LIN {X 0,Y 162.207,Z 623.007,A -85,B 0,C 180,E1 -23497.47,E2 -23497.47} C_VEL
LIN {X 0,Y 162.719,Z 622.375,A -85,B 0,C 180,E1 -23499.95,E2 -23499.95} C_VEL
LIN {X 0,Y 163.523,Z 621.28,A -85,B 0,C 180,E1 -23502.411,E2 -23502.411} C_VEL
LIN {X 0,Y 165.346,Z 618.557,A -85,B 0,C 180,E1 -23506.04,E2 -23506.04} C_VEL
LIN {X 0,Y 167.897,Z 614.612,A -85,B 0,C 180,E1 -23509.566,E2 -23509.566} C_VEL
LIN {X 0,Y 168.435,Z 613.877,A -85,B 0,C 180,E1 -23510.136,E2 -23510.136} C_VEL
LIN {X 0,Y 170.028,Z 614.229,A -85,B 0,C 180,E1 -23511.925,E2 -23511.925} C_VEL
LIN {X 0,Y 175.274,Z 613.945,A -85,B 0,C 180,E1 -23516.173,E2 -23516.173} C_VEL
LIN {X 0,Y 178.341,Z 613.349,A -85,B 0,C 180,E1 -23518.223,E2 -23518.223} C_VEL
LIN {X 0,Y 183.249,Z 611.746,A -85,B 0,C 180,E1 -23520.885,E2 -23520.885} C_VEL
LIN {X 0,Y 185.044,Z 611.049,A -85,B 0,C 180,E1 -23521.95,E2 -23521.95} C_VEL
LIN {X 0,Y 186.792,Z 609.893,A -85,B 0,C 180,E1 -23523.665,E2 -23523.665} C_VEL
LIN {X 0,Y 188.276,Z 608.112,A -85,B 0,C 180,E1 -23526.659,E2 -23526.659} C_VEL
LIN {X 0,Y 190.28,Z 605.857,A -85,B 0,C 180,E1 -23530.266,E2 -23530.266} C_VEL
LIN {X 0,Y 191.354,Z 605.077,A -85,B 0,C 180,E1 -23531.385,E2 -23531.385} C_VEL
LIN {X 0,Y 192.086,Z 604.286,A -85,B 0,C 180,E1 -23532.966,E2 -23532.966} C_VEL
LIN {X 0,Y 192.613,Z 603.111,A -85,B 0,C 180,E1 -23536.867,E2 -23536.867} C_VEL
LIN {X 0,Y 192.568,Z 602.746,A -85,B 0,C 180,E1 -23540.035,E2 -23540.035} C_VEL
LIN {X 0,Y 192.239,Z 602.8,A -85,B 0,C 180,E1 -23541.575,E2 -23541.575} C_VEL
LIN {X 0,Y 191.24,Z 603.167,A -85,B 0,C 180,E1 -23543.985,E2 -23543.985} C_VEL
LIN {X 0,Y 188.877,Z 604.094,A -85,B 0,C 180,E1 -23546.073,E2 -23546.073} C_VEL
LIN {X 0,Y 184.48,Z 605.231,A -85,B 0,C 180,E1 -23547.768,E2 -23547.768} C_VEL
LIN {X 0,Y 176.516,Z 606.429,A -85,B 0,C 180,E1 -23551.46,E2 -23551.46} C_VEL
LIN {X 0,Y 171.67,Z 606.356,A -85,B 0,C 180,E1 -23554.248,E2 -23554.248} C_VEL
LIN {X 0,Y 166.772,Z 605.292,A -85,B 0,C 180,E1 -23557.712,E2 -23557.712} C_VEL
LIN {X 0,Y 164.167,Z 604.166,A -85,B 0,C 180,E1 -23559.972,E2 -23559.972} C_VEL
LIN {X 0,Y 159.875,Z 600.675,A -85,B 0,C 180,E1 -23564.707,E2 -23564.707} C_VEL
LIN {X 0,Y 157.891,Z 597.165,A -85,B 0,C 180,E1 -23568.315,E2 -23568.315} C_VEL
LIN {X 0,Y 156.697,Z 592.416,A -85,B 0,C 180,E1 -23572.267,E2 -23572.267} C_VEL
LIN {X 0,Y 156.112,Z 586.613,A -85,B 0,C 180,E1 -23576.128,E2 -23576.128} C_VEL
LIN {X 0,Y 156.043,Z 579.511,A -85,B 0,C 180,E1 -23580,E2 -23580} C_VEL
LIN {X 0,Y 156.277,Z 572.106,A -85,B 0,C 180,E1 -23583.223,E2 -23583.223} C_VEL
LIN {X 0,Y 156.781,Z 562.966,A -85,B 0,C 180,E1 -23586.435,E2 -23586.435} C_VEL
LIN {X 0,Y 156.964,Z 559.635,A -85,B 0,C 180,E1 -23587.477,E2 -23587.477} C_VEL
LIN {X 0,Y 156.789,Z 560.465,A -85,B 0,C 180,E1 -23587.728,E2 -23587.728} C_VEL
LIN {X 0,Y 158.13,Z 562.339,A -85,B 0,C 180,E1 -23589.28,E2 -23589.28} C_VEL
LIN {X 0,Y 160.819,Z 561.897,A -85,B 0,C 180,E1 -23590.717,E2 -23590.717} C_VEL
LIN {X 0,Y 163.892,Z 561.849,A -85,B 0,C 180,E1 -23592.381,E2 -23592.381} C_VEL
LIN {X 0,Y 168.567,Z 561.369,A -85,B 0,C 180,E1 -23594.487,E2 -23594.487} C_VEL
LIN {X 0,Y 172.959,Z 561.867,A -85,B 0,C 180,E1 -23596.525,E2 -23596.525} C_VEL
LIN {X 0,Y 175.402,Z 568.322,A -85,B 0,C 180,E1 -23599.303,E2 -23599.303} C_VEL
LIN {X 0,Y 175.617,Z 573.789,A -85,B 0,C 180,E1 -23601.111,E2 -23601.111} C_VEL
LIN {X 0,Y 175.037,Z 581.344,A -85,B 0,C 180,E1 -23603.673,E2 -23603.673} C_VEL
LIN {X 0,Y 174.064,Z 586.458,A -85,B 0,C 180,E1 -23605.485,E2 -23605.485} C_VEL
LIN {X 0,Y 170.852,Z 593.117,A -85,B 0,C 180,E1 -23607.82,E2 -23607.82} C_VEL
LIN {X 0,Y 167.861,Z 598.504,A -85,B 0,C 180,E1 -23610.16,E2 -23610.16} C_VEL
LIN {X 0,Y 164.679,Z 603.67,A -85,B 0,C 180,E1 -23613.039,E2 -23613.039} C_VEL
LIN {X 0,Y 161.608,Z 608.225,A -85,B 0,C 180,E1 -23616.436,E2 -23616.436} C_VEL
LIN {X 0,Y 159.378,Z 611.17,A -85,B 0,C 180,E1 -23619.492,E2 -23619.492} C_VEL
LIN {X 0,Y 157.997,Z 612.779,A -85,B 0,C 180,E1 -23621.854,E2 -23621.854} C_VEL
LIN {X 0,Y 156.118,Z 614.605,A -85,B 0,C 180,E1 -23626.077,E2 -23626.077} C_VEL
LIN {X 0,Y 154.878,Z 614.948,A -85,B 0,C 180,E1 -23630.557,E2 -23630.557} C_VEL
LIN {X 0,Y 154.344,Z 613.836,A -85,B 0,C 180,E1 -23635.047,E2 -23635.047} C_VEL
LIN {X 0,Y 154.333,Z 612.995,A -85,B 0,C 180,E1 -23636.874,E2 -23636.874} C_VEL
LIN {X 0,Y 154.603,Z 610.912,A -85,B 0,C 180,E1 -23639.996,E2 -23639.996} C_VEL
LIN {X 0,Y 155.155,Z 608.065,A -85,B 0,C 180,E1 -23643.064,E2 -23643.064} C_VEL
LIN {X 0,Y 156.072,Z 603.34,A -85,B 0,C 180,E1 -23646.794,E2 -23646.794} C_VEL
LIN {X 0,Y 157.166,Z 598.254,A -85,B 0,C 180,E1 -23649.894,E2 -23649.894} C_VEL
LIN {X 0,Y 158.396,Z 592.777,A -85,B 0,C 180,E1 -23652.571,E2 -23652.571} C_VEL
LIN {X 0,Y 160.251,Z 585.018,A -85,B 0,C 180,E1 -23655.611,E2 -23655.611} C_VEL
LIN {X 0,Y 162.014,Z 576.781,A -85,B 0,C 180,E1 -23658.108,E2 -23658.108} C_VEL
LIN {X 0,Y 162.751,Z 572.847,A -85,B 0,C 180,E1 -23659.109,E2 -23659.109} C_VEL
LIN {X 0,Y 162.183,Z 562.521,A -85,B 0,C 180,E1 -23661.589,E2 -23661.589} C_VEL
LIN {X 0,Y 161.198,Z 552.872,A -85,B 0,C 180,E1 -23663.427,E2 -23663.427} C_VEL
LIN {X 0,Y 159.728,Z 543.138,A -85,B 0,C 180,E1 -23664.95,E2 -23664.95} C_VEL
LIN {X 0,Y 157.671,Z 532.624,A -85,B 0,C 180,E1 -23666.325,E2 -23666.325} C_VEL
LIN {X 0,Y 158.334,Z 527.356,A -85,B 0,C 180,E1 -23671.27,E2 -23671.27} C_VEL
LIN {X 0,Y 157.895,Z 525.63,A -85,B 0,C 180,E1 -23673.188,E2 -23673.188} C_VEL
LIN {X 0,Y 157.826,Z 525.639,A -85,B 0,C 180,E1 -23677.676,E2 -23677.676} C_VEL
LIN {X 0,Y 157.707,Z 525.652,A -85,B 0,C 180,E1 -23681.361,E2 -23681.361} C_VEL
LIN {X 0,Y 157.479,Z 525.68,A -85,B 0,C 180,E1 -23685.53,E2 -23685.53} C_VEL
LIN {X 0,Y 157.37,Z 525.693,A -85,B 0,C 180,E1 -23690.931,E2 -23690.931} C_VEL
LIN {X 0,Y 157.315,Z 525.701,A -85,B 0,C 180,E1 -23696.684,E2 -23696.684} C_VEL
LIN {X 0,Y 157.278,Z 525.705,A -85,B 0,C 180,E1 -23702.425,E2 -23702.425} C_VEL
LIN {X 0,Y 157.317,Z 525.701,A -85,B 0,C 180,E1 -23706.473,E2 -23706.473} C_VEL
LIN {X 0,Y 157.274,Z 525.7,A -85,B 0,C 180,E1 -23712.088,E2 -23712.088} C_VEL
LIN {X 0,Y 157.3,Z 525.701,A -85,B 0,C 180,E1 -23715.63,E2 -23715.63} C_VEL
LIN {X 0,Y 157.285,Z 525.7,A -85,B 0,C 180,E1 -23721.276,E2 -23721.276} C_VEL
LIN {X 0,Y 157.29,Z 525.698,A -85,B 0,C 180,E1 -23724.488,E2 -23724.488} C_VEL
LIN {X 0,Y 157.291,Z 525.706,A -85,B 0,C 180,E1 -23728.095,E2 -23728.095} C_VEL
LIN {X 0,Y 157.319,Z 525.696,A -85,B 0,C 180,E1 -23733.465,E2 -23733.465} C_VEL
LIN {X 0,Y 157.392,Z 525.69,A -85,B 0,C 180,E1 -23739.667,E2 -23739.667} C_VEL
LIN {X 0,Y 157.476,Z 525.681,A -85,B 0,C 180,E1 -23744.468,E2 -23744.468} C_VEL
LIN {X 0,Y 157.77,Z 525.641,A -85,B 0,C 180,E1 -23749.736,E2 -23749.736} C_VEL
LIN {X 0,Y 157.822,Z 525.638,A -85,B 0,C 180,E1 -23752.323,E2 -23752.323} C_VEL
LIN {X 0,Y 158.256,Z 525.576,A -85,B 0,C 180,E1 -23760,E2 -23760} C_VEL
LIN {X 0,Y 157.822,Z 525.637,A -85,B 0,C 180,E1 -23767.677,E2 -23767.677} C_VEL
LIN {X 0,Y 157.703,Z 525.654,A -85,B 0,C 180,E1 -23771.362,E2 -23771.362} C_VEL
LIN {X 0,Y 157.476,Z 525.684,A -85,B 0,C 180,E1 -23775.532,E2 -23775.532} C_VEL
LIN {X 0,Y 157.367,Z 525.695,A -85,B 0,C 180,E1 -23780.933,E2 -23780.933} C_VEL
LIN {X 0,Y 157.312,Z 525.704,A -85,B 0,C 180,E1 -23786.685,E2 -23786.685} C_VEL
LIN {X 0,Y 157.276,Z 525.707,A -85,B 0,C 180,E1 -23792.427,E2 -23792.427} C_VEL
LIN {X 0,Y 157.281,Z 525.704,A -85,B 0,C 180,E1 -23796.458,E2 -23796.458} C_VEL
LIN {X 0,Y 157.23,Z 525.714,A -85,B 0,C 180,E1 -23802.104,E2 -23802.104} C_VEL
LIN {X 0,Y 157.323,Z 525.701,A -85,B 0,C 180,E1 -23807.928,E2 -23807.928} C_VEL
LIN {X 0,Y 157.937,Z 525.823,A -85,B 0,C 180,E1 -23814.498,E2 -23814.498} C_VEL
LIN {X 0,Y 158.756,Z 528.891,A -85,B 0,C 180,E1 -23816.218,E2 -23816.218} C_VEL
LIN {X 0,Y 158.764,Z 532.311,A -85,B 0,C 180,E1 -23817.915,E2 -23817.915} C_VEL
LIN {X 0,Y 158.394,Z 536.375,A -85,B 0,C 180,E1 -23819.811,E2 -23819.811} C_VEL
LIN {X 0,Y 160.336,Z 549.59,A -85,B 0,C 180,E1 -23821.175,E2 -23821.175} C_VEL
LIN {X 0,Y 161.128,Z 558.733,A -85,B 0,C 180,E1 -23822.41,E2 -23822.41} C_VEL
LIN {X 0,Y 161.352,Z 567.841,A -85,B 0,C 180,E1 -23823.926,E2 -23823.926} C_VEL
LIN {X 0,Y 161.312,Z 576.509,A -85,B 0,C 180,E1 -23825.715,E2 -23825.715} C_VEL
LIN {X 0,Y 160.941,Z 586.296,A -85,B 0,C 180,E1 -23828.213,E2 -23828.213} C_VEL
LIN {X 0,Y 159.369,Z 594.146,A -85,B 0,C 180,E1 -23830.688,E2 -23830.688} C_VEL
LIN {X 0,Y 157.885,Z 600.548,A -85,B 0,C 180,E1 -23833.183,E2 -23833.183} C_VEL
LIN {X 0,Y 156.793,Z 605.878,A -85,B 0,C 180,E1 -23835.729,E2 -23835.729} C_VEL
LIN {X 0,Y 155.929,Z 610.305,A -85,B 0,C 180,E1 -23838.299,E2 -23838.299} C_VEL
LIN {X 0,Y 155.113,Z 615.472,A -85,B 0,C 180,E1 -23842.189,E2 -23842.189} C_VEL
LIN {X 0,Y 154.855,Z 618.102,A -85,B 0,C 180,E1 -23844.793,E2 -23844.793} C_VEL
LIN {X 0,Y 154.815,Z 620.154,A -85,B 0,C 180,E1 -23847.399,E2 -23847.399} C_VEL
LIN {X 0,Y 154.892,Z 621.665,A -85,B 0,C 180,E1 -23850.001,E2 -23850.001} C_VEL
LIN {X 0,Y 154.775,Z 622.571,A -85,B 0,C 180,E1 -23852.604,E2 -23852.604} C_VEL
LIN {X 0,Y 154.857,Z 622.945,A -85,B 0,C 180,E1 -23855.209,E2 -23855.209} C_VEL
LIN {X 0,Y 155.172,Z 622.861,A -85,B 0,C 180,E1 -23857.811,E2 -23857.811} C_VEL
LIN {X 0,Y 155.715,Z 622.321,A -85,B 0,C 180,E1 -23860.402,E2 -23860.402} C_VEL
LIN {X 0,Y 156.597,Z 621.297,A -85,B 0,C 180,E1 -23862.969,E2 -23862.969} C_VEL
LIN {X 0,Y 158.528,Z 618.696,A -85,B 0,C 180,E1 -23866.749,E2 -23866.749} C_VEL
LIN {X 0,Y 161.228,Z 614.868,A -85,B 0,C 180,E1 -23870.411,E2 -23870.411} C_VEL
LIN {X 0,Y 162.615,Z 613.157,A -85,B 0,C 180,E1 -23871.887,E2 -23871.887} C_VEL
LIN {X 0,Y 166.021,Z 613.673,A -85,B 0,C 180,E1 -23875.046,E2 -23875.046} C_VEL
LIN {X 0,Y 168.934,Z 613.649,A -85,B 0,C 180,E1 -23877.235,E2 -23877.235} C_VEL
LIN {X 0,Y 175.704,Z 612.497,A -85,B 0,C 180,E1 -23881.333,E2 -23881.333} C_VEL
LIN {X 0,Y 179.68,Z 611.368,A -85,B 0,C 180,E1 -23883.203,E2 -23883.203} C_VEL
LIN {X 0,Y 183.551,Z 609.907,A -85,B 0,C 180,E1 -23885.054,E2 -23885.054} C_VEL
LIN {X 0,Y 186.575,Z 608.394,A -85,B 0,C 180,E1 -23887.065,E2 -23887.065} C_VEL
LIN {X 0,Y 189.284,Z 606.633,A -85,B 0,C 180,E1 -23889.14,E2 -23889.14} C_VEL
LIN {X 0,Y 190.28,Z 605.857,A -85,B 0,C 180,E1 -23890.266,E2 -23890.266} C_VEL
LIN {X 0,Y 190.856,Z 605.242,A -85,B 0,C 180,E1 -23891.41,E2 -23891.41} C_VEL
LIN {X 0,Y 190.445,Z 604.805,A -85,B 0,C 180,E1 -23893.173,E2 -23893.173} C_VEL
LIN {X 0,Y 189.135,Z 604.766,A -85,B 0,C 180,E1 -23894.933,E2 -23894.933} C_VEL
LIN {X 0,Y 186.189,Z 605.068,A -85,B 0,C 180,E1 -23898.626,E2 -23898.626} C_VEL
LIN {X 0,Y 185.854,Z 605.035,A -85,B 0,C 180,E1 -23899.895,E2 -23899.895} C_VEL
LIN {X 0,Y 184.79,Z 605.138,A -85,B 0,C 180,E1 -23903.006,E2 -23903.006} C_VEL
LIN {X 0,Y 182.966,Z 605.531,A -85,B 0,C 180,E1 -23904.818,E2 -23904.818} C_VEL
LIN {X 0,Y 174.336,Z 606.945,A -85,B 0,C 180,E1 -23908.395,E2 -23908.395} C_VEL
LIN {X 0,Y 166.248,Z 606.681,A -85,B 0,C 180,E1 -23912.596,E2 -23912.596} C_VEL
LIN {X 0,Y 163.292,Z 606.167,A -85,B 0,C 180,E1 -23914.508,E2 -23914.508} C_VEL
LIN {X 0,Y 157.542,Z 603.712,A -85,B 0,C 180,E1 -23919.091,E2 -23919.091} C_VEL
LIN {X 0,Y 154.115,Z 600.908,A -85,B 0,C 180,E1 -23922.758,E2 -23922.758} C_VEL
LIN {X 0,Y 151.609,Z 597.215,A -85,B 0,C 180,E1 -23926.598,E2 -23926.598} C_VEL
LIN {X 0,Y 150.168,Z 592.578,A -85,B 0,C 180,E1 -23930.572,E2 -23930.572} C_VEL
LIN {X 0,Y 149.434,Z 586.884,A -85,B 0,C 180,E1 -23934.603,E2 -23934.603} C_VEL
LIN {X 0,Y 149.186,Z 579.766,A -85,B 0,C 180,E1 -23938.651,E2 -23938.651} C_VEL
LIN {X 0,Y 149.403,Z 572.526,A -85,B 0,C 180,E1 -23942.022,E2 -23942.022} C_VEL
LIN {X 0,Y 149.647,Z 565.842,A -85,B 0,C 180,E1 -23944.63,E2 -23944.63} C_VEL
LIN {X 0,Y 149.485,Z 567.428,A -85,B 0,C 180,E1 -23945.396,E2 -23945.396} C_VEL
LIN {X 0,Y 152.87,Z 567.395,A -85,B 0,C 180,E1 -23947.928,E2 -23947.928} C_VEL
LIN {X 0,Y 155.992,Z 568.381,A -85,B 0,C 180,E1 -23950.382,E2 -23950.382} C_VEL
LIN {X 0,Y 164.946,Z 567.632,A -85,B 0,C 180,E1 -23954.812,E2 -23954.812} C_VEL
LIN {X 0,Y 168.848,Z 568.796,A -85,B 0,C 180,E1 -23956.94,E2 -23956.94} C_VEL
LIN {X 0,Y 170.034,Z 572.646,A -85,B 0,C 180,E1 -23958.683,E2 -23958.683} C_VEL
LIN {X 0,Y 169.597,Z 579.862,A -85,B 0,C 180,E1 -23961.26,E2 -23961.26} C_VEL
LIN {X 0,Y 168.174,Z 587.363,A -85,B 0,C 180,E1 -23964.13,E2 -23964.13} C_VEL
LIN {X 0,Y 164.933,Z 593.81,A -85,B 0,C 180,E1 -23966.51,E2 -23966.51} C_VEL
LIN {X 0,Y 161.238,Z 599.946,A -85,B 0,C 180,E1 -23969.334,E2 -23969.334} C_VEL
LIN {X 0,Y 157.228,Z 605.949,A -85,B 0,C 180,E1 -23973.056,E2 -23973.056} C_VEL
LIN {X 0,Y 154.425,Z 609.605,A -85,B 0,C 180,E1 -23976.274,E2 -23976.274} C_VEL
LIN {X 0,Y 152.748,Z 611.555,A -85,B 0,C 180,E1 -23978.538,E2 -23978.538} C_VEL
LIN {X 0,Y 150.822,Z 613.566,A -85,B 0,C 180,E1 -23981.79,E2 -23981.79} C_VEL
LIN {X 0,Y 149.331,Z 614.771,A -85,B 0,C 180,E1 -23985.092,E2 -23985.092} C_VEL
LIN {X 0,Y 147.999,Z 615.206,A -85,B 0,C 180,E1 -23989.446,E2 -23989.446} C_VEL
LIN {X 0,Y 147.303,Z 614.173,A -85,B 0,C 180,E1 -23994.203,E2 -23994.203} C_VEL
LIN {X 0,Y 147.373,Z 611.609,A -85,B 0,C 180,E1 -23999.137,E2 -23999.137} C_VEL
LIN {X 0,Y 148.04,Z 608.225,A -85,B 0,C 180,E1 -24003.026,E2 -24003.026} C_VEL
LIN {X 0,Y 149.03,Z 603.251,A -85,B 0,C 180,E1 -24007.103,E2 -24007.103} C_VEL
LIN {X 0,Y 150.148,Z 598.211,A -85,B 0,C 180,E1 -24010.283,E2 -24010.283} C_VEL
LIN {X 0,Y 151.466,Z 592.563,A -85,B 0,C 180,E1 -24013.141,E2 -24013.141} C_VEL
LIN {X 0,Y 153.372,Z 584.895,A -85,B 0,C 180,E1 -24016.242,E2 -24016.242} C_VEL
LIN {X 0,Y 155.287,Z 576.297,A -85,B 0,C 180,E1 -24018.909,E2 -24018.909} C_VEL
LIN {X 0,Y 155.824,Z 572.513,A -85,B 0,C 180,E1 -24019.933,E2 -24019.933} C_VEL
LIN {X 0,Y 155.241,Z 561.98,A -85,B 0,C 180,E1 -24022.52,E2 -24022.52} C_VEL
LIN {X 0,Y 154.221,Z 552.27,A -85,B 0,C 180,E1 -24024.442,E2 -24024.442} C_VEL
LIN {X 0,Y 152.614,Z 541.928,A -85,B 0,C 180,E1 -24026.12,E2 -24026.12} C_VEL
LIN {X 0,Y 150.798,Z 532.806,A -85,B 0,C 180,E1 -24027.327,E2 -24027.327} C_VEL
LIN {X 0,Y 151.343,Z 528.659,A -85,B 0,C 180,E1 -24031.329,E2 -24031.329} C_VEL
LIN {X 0,Y 150.826,Z 526.51,A -85,B 0,C 180,E1 -24033.672,E2 -24033.672} C_VEL
LIN {X 0,Y 150.765,Z 526.519,A -85,B 0,C 180,E1 -24038.038,E2 -24038.038} C_VEL
LIN {X 0,Y 150.636,Z 526.533,A -85,B 0,C 180,E1 -24041.545,E2 -24041.545} C_VEL
LIN {X 0,Y 150.384,Z 526.564,A -85,B 0,C 180,E1 -24046.283,E2 -24046.283} C_VEL
LIN {X 0,Y 150.351,Z 526.567,A -85,B 0,C 180,E1 -24050.791,E2 -24050.791} C_VEL
LIN {X 0,Y 150.244,Z 526.581,A -85,B 0,C 180,E1 -24057.281,E2 -24057.281} C_VEL
LIN {X 0,Y 150.218,Z 526.584,A -85,B 0,C 180,E1 -24062.633,E2 -24062.633} C_VEL
LIN {X 0,Y 150.223,Z 526.584,A -85,B 0,C 180,E1 -24067.457,E2 -24067.457} C_VEL
LIN {X 0,Y 150.21,Z 526.582,A -85,B 0,C 180,E1 -24071.53,E2 -24071.53} C_VEL
LIN {X 0,Y 150.249,Z 526.578,A -85,B 0,C 180,E1 -24075.441,E2 -24075.441} C_VEL
LIN {X 0,Y 150.228,Z 526.582,A -85,B 0,C 180,E1 -24079.084,E2 -24079.084} C_VEL
LIN {X 0,Y 150.234,Z 526.572,A -85,B 0,C 180,E1 -24082.678,E2 -24082.678} C_VEL
LIN {X 0,Y 150.215,Z 526.584,A -85,B 0,C 180,E1 -24087.365,E2 -24087.365} C_VEL
LIN {X 0,Y 150.242,Z 526.576,A -85,B 0,C 180,E1 -24092.717,E2 -24092.717} C_VEL
LIN {X 0,Y 150.349,Z 526.567,A -85,B 0,C 180,E1 -24099.207,E2 -24099.207} C_VEL
LIN {X 0,Y 150.381,Z 526.565,A -85,B 0,C 180,E1 -24103.715,E2 -24103.715} C_VEL
LIN {X 0,Y 150.687,Z 526.521,A -85,B 0,C 180,E1 -24109.248,E2 -24109.248} C_VEL
LIN {X 0,Y 150.761,Z 526.519,A -85,B 0,C 180,E1 -24111.961,E2 -24111.961} C_VEL
LIN {X 0,Y 151.216,Z 526.452,A -85,B 0,C 180,E1 -24120,E2 -24120} C_VEL
LIN {X 0,Y 150.761,Z 526.518,A -85,B 0,C 180,E1 -24128.039,E2 -24128.039} C_VEL
LIN {X 0,Y 150.632,Z 526.534,A -85,B 0,C 180,E1 -24131.546,E2 -24131.546} C_VEL
LIN {X 0,Y 150.38,Z 526.564,A -85,B 0,C 180,E1 -24136.284,E2 -24136.284} C_VEL
LIN {X 0,Y 150.348,Z 526.57,A -85,B 0,C 180,E1 -24140.793,E2 -24140.793} C_VEL
LIN {X 0,Y 150.242,Z 526.586,A -85,B 0,C 180,E1 -24147.283,E2 -24147.283} C_VEL
LIN {X 0,Y 150.216,Z 526.586,A -85,B 0,C 180,E1 -24152.635,E2 -24152.635} C_VEL
LIN {X 0,Y 150.209,Z 526.585,A -85,B 0,C 180,E1 -24157.462,E2 -24157.462} C_VEL
LIN {X 0,Y 150.168,Z 526.592,A -85,B 0,C 180,E1 -24161.514,E2 -24161.514} C_VEL
LIN {X 0,Y 150.189,Z 526.59,A -85,B 0,C 180,E1 -24165.421,E2 -24165.421} C_VEL
LIN {X 0,Y 150.332,Z 526.572,A -85,B 0,C 180,E1 -24169.12,E2 -24169.12} C_VEL
LIN {X 0,Y 150.773,Z 526.721,A -85,B 0,C 180,E1 -24173.538,E2 -24173.538} C_VEL
LIN {X 0,Y 151.819,Z 529.881,A -85,B 0,C 180,E1 -24175.455,E2 -24175.455} C_VEL
LIN {X 0,Y 151.937,Z 533.352,A -85,B 0,C 180,E1 -24177.307,E2 -24177.307} C_VEL
LIN {X 0,Y 151.634,Z 536.634,A -85,B 0,C 180,E1 -24178.833,E2 -24178.833} C_VEL
LIN {X 0,Y 153.5,Z 549.179,A -85,B 0,C 180,E1 -24180.19,E2 -24180.19} C_VEL
LIN {X 0,Y 154.308,Z 558.245,A -85,B 0,C 180,E1 -24181.477,E2 -24181.477} C_VEL
LIN {X 0,Y 154.489,Z 566.777,A -85,B 0,C 180,E1 -24182.942,E2 -24182.942} C_VEL
LIN {X 0,Y 154.475,Z 575.328,A -85,B 0,C 180,E1 -24184.756,E2 -24184.756} C_VEL
LIN {X 0,Y 154.186,Z 583.468,A -85,B 0,C 180,E1 -24186.852,E2 -24186.852} C_VEL
LIN {X 0,Y 153.763,Z 588.024,A -85,B 0,C 180,E1 -24188.202,E2 -24188.202} C_VEL
LIN {X 0,Y 152.226,Z 594.656,A -85,B 0,C 180,E1 -24190.446,E2 -24190.446} C_VEL
LIN {X 0,Y 150.759,Z 600.942,A -85,B 0,C 180,E1 -24193.062,E2 -24193.062} C_VEL
LIN {X 0,Y 149.64,Z 606.165,A -85,B 0,C 180,E1 -24195.727,E2 -24195.727} C_VEL
LIN {X 0,Y 148.601,Z 611.45,A -85,B 0,C 180,E1 -24199.097,E2 -24199.097} C_VEL
LIN {X 0,Y 148.06,Z 614.836,A -85,B 0,C 180,E1 -24201.815,E2 -24201.815} C_VEL
LIN {X 0,Y 147.79,Z 617.574,A -85,B 0,C 180,E1 -24204.544,E2 -24204.544} C_VEL
LIN {X 0,Y 147.719,Z 619.902,A -85,B 0,C 180,E1 -24207.581,E2 -24207.581} C_VEL
LIN {X 0,Y 147.796,Z 621.288,A -85,B 0,C 180,E1 -24210.001,E2 -24210.001} C_VEL
LIN {X 0,Y 147.695,Z 622.238,A -85,B 0,C 180,E1 -24212.729,E2 -24212.729} C_VEL
LIN {X 0,Y 147.792,Z 622.705,A -85,B 0,C 180,E1 -24215.459,E2 -24215.459} C_VEL
LIN {X 0,Y 148.119,Z 622.714,A -85,B 0,C 180,E1 -24218.185,E2 -24218.185} C_VEL
LIN {X 0,Y 148.734,Z 622.269,A -85,B 0,C 180,E1 -24220.896,E2 -24220.896} C_VEL
LIN {X 0,Y 149.694,Z 621.277,A -85,B 0,C 180,E1 -24223.578,E2 -24223.578} C_VEL
LIN {X 0,Y 151.743,Z 618.862,A -85,B 0,C 180,E1 -24227.522,E2 -24227.522} C_VEL
LIN {X 0,Y 154.597,Z 615.157,A -85,B 0,C 180,E1 -24231.328,E2 -24231.328} C_VEL
LIN {X 0,Y 156.803,Z 612.376,A -85,B 0,C 180,E1 -24233.616,E2 -24233.616} C_VEL
LIN {X 0,Y 162.686,Z 613.083,A -85,B 0,C 180,E1 -24238.374,E2 -24238.374} C_VEL
LIN {X 0,Y 165.992,Z 613.004,A -85,B 0,C 180,E1 -24240.537,E2 -24240.537} C_VEL
LIN {X 0,Y 173.805,Z 611.628,A -85,B 0,C 180,E1 -24244.481,E2 -24244.481} C_VEL
LIN {X 0,Y 177.724,Z 610.529,A -85,B 0,C 180,E1 -24246.383,E2 -24246.383} C_VEL
LIN {X 0,Y 182.416,Z 608.388,A -85,B 0,C 180,E1 -24249.597,E2 -24249.597} C_VEL
LIN {X 0,Y 183.587,Z 607.718,A -85,B 0,C 180,E1 -24250.786,E2 -24250.786} C_VEL
LIN {X 0,Y 185.295,Z 606.516,A -85,B 0,C 180,E1 -24253.058,E2 -24253.058} C_VEL
LIN {X 0,Y 185.911,Z 605.372,A -85,B 0,C 180,E1 -24257.121,E2 -24257.121} C_VEL
LIN {X 0,Y 185.854,Z 605.035,A -85,B 0,C 180,E1 -24259.895,E2 -24259.895} C_VEL
LIN {X 0,Y 185.169,Z 605.186,A -85,B 0,C 180,E1 -24260.858,E2 -24260.858} C_VEL
LIN {X 0,Y 182.748,Z 605.725,A -85,B 0,C 180,E1 -24262.057,E2 -24262.057} C_VEL
LIN {X 0,Y 176.733,Z 606.906,A -85,B 0,C 180,E1 -24263.881,E2 -24263.881} C_VEL
LIN {X 0,Y 172.841,Z 607.378,A -85,B 0,C 180,E1 -24265.235,E2 -24265.235} C_VEL
LIN {X 0,Y 164.22,Z 607.472,A -85,B 0,C 180,E1 -24269.099,E2 -24269.099} C_VEL
LIN {X 0,Y 160.388,Z 606.91,A -85,B 0,C 180,E1 -24271.184,E2 -24271.184} C_VEL
LIN {X 0,Y 153.763,Z 604.776,A -85,B 0,C 180,E1 -24275.71,E2 -24275.71} C_VEL
LIN {X 0,Y 148.558,Z 601.086,A -85,B 0,C 180,E1 -24280.661,E2 -24280.661} C_VEL
LIN {X 0,Y 145.567,Z 597.317,A -85,B 0,C 180,E1 -24284.601,E2 -24284.601} C_VEL
LIN {X 0,Y 143.733,Z 592.677,A -85,B 0,C 180,E1 -24288.721,E2 -24288.721} C_VEL
LIN {X 0,Y 142.701,Z 585.937,A -85,B 0,C 180,E1 -24293.638,E2 -24293.638} C_VEL
LIN {X 0,Y 142.399,Z 578.623,A -85,B 0,C 180,E1 -24297.879,E2 -24297.879} C_VEL
LIN {X 0,Y 142.586,Z 571.267,A -85,B 0,C 180,E1 -24301.412,E2 -24301.412} C_VEL
LIN {X 0,Y 142.309,Z 572.695,A -85,B 0,C 180,E1 -24302.123,E2 -24302.123} C_VEL
LIN {X 0,Y 142.597,Z 573.283,A -85,B 0,C 180,E1 -24302.825,E2 -24302.825} C_VEL
LIN {X 0,Y 149.166,Z 573.401,A -85,B 0,C 180,E1 -24308.332,E2 -24308.332} C_VEL
LIN {X 0,Y 152.028,Z 574.208,A -85,B 0,C 180,E1 -24310.656,E2 -24310.656} C_VEL
LIN {X 0,Y 160.894,Z 573.677,A -85,B 0,C 180,E1 -24315.194,E2 -24315.194} C_VEL
LIN {X 0,Y 164.234,Z 575.396,A -85,B 0,C 180,E1 -24317.431,E2 -24317.431} C_VEL
LIN {X 0,Y 164.21,Z 578.6,A -85,B 0,C 180,E1 -24318.724,E2 -24318.724} C_VEL
LIN {X 0,Y 163.125,Z 585.576,A -85,B 0,C 180,E1 -24321.482,E2 -24321.482} C_VEL
LIN {X 0,Y 161.692,Z 590.106,A -85,B 0,C 180,E1 -24323.358,E2 -24323.358} C_VEL
LIN {X 0,Y 157.075,Z 597.881,A -85,B 0,C 180,E1 -24326.579,E2 -24326.579} C_VEL
LIN {X 0,Y 153.408,Z 603.104,A -85,B 0,C 180,E1 -24329.488,E2 -24329.488} C_VEL
LIN {X 0,Y 150.18,Z 607.326,A -85,B 0,C 180,E1 -24332.609,E2 -24332.609} C_VEL
LIN {X 0,Y 147.386,Z 610.581,A -85,B 0,C 180,E1 -24335.84,E2 -24335.84} C_VEL
LIN {X 0,Y 145.051,Z 612.948,A -85,B 0,C 180,E1 -24339.172,E2 -24339.172} C_VEL
LIN {X 0,Y 142.77,Z 614.807,A -85,B 0,C 180,E1 -24343.564,E2 -24343.564} C_VEL
LIN {X 0,Y 141.147,Z 615.437,A -85,B 0,C 180,E1 -24348.321,E2 -24348.321} C_VEL
LIN {X 0,Y 140.263,Z 614.499,A -85,B 0,C 180,E1 -24353.292,E2 -24353.292} C_VEL
LIN {X 0,Y 140.216,Z 612.059,A -85,B 0,C 180,E1 -24358.44,E2 -24358.44} C_VEL
LIN {X 0,Y 140.995,Z 608.003,A -85,B 0,C 180,E1 -24363.344,E2 -24363.344} C_VEL
LIN {X 0,Y 141.967,Z 603.235,A -85,B 0,C 180,E1 -24367.387,E2 -24367.387} C_VEL
LIN {X 0,Y 143.433,Z 596.967,A -85,B 0,C 180,E1 -24371.427,E2 -24371.427} C_VEL
LIN {X 0,Y 145.371,Z 589.045,A -85,B 0,C 180,E1 -24375.219,E2 -24375.219} C_VEL
LIN {X 0,Y 146.893,Z 582.888,A -85,B 0,C 180,E1 -24377.566,E2 -24377.566} C_VEL
LIN {X 0,Y 148.575,Z 575.782,A -85,B 0,C 180,E1 -24379.781,E2 -24379.781} C_VEL
LIN {X 0,Y 148.877,Z 572.166,A -85,B 0,C 180,E1 -24380.831,E2 -24380.831} C_VEL
LIN {X 0,Y 148.337,Z 561.441,A -85,B 0,C 180,E1 -24383.538,E2 -24383.538} C_VEL
LIN {X 0,Y 147.291,Z 551.674,A -85,B 0,C 180,E1 -24385.552,E2 -24385.552} C_VEL
LIN {X 0,Y 145.834,Z 542.262,A -85,B 0,C 180,E1 -24387.15,E2 -24387.15} C_VEL
LIN {X 0,Y 143.943,Z 532.86,A -85,B 0,C 180,E1 -24388.512,E2 -24388.512} C_VEL
LIN {X 0,Y 144.349,Z 529.994,A -85,B 0,C 180,E1 -24391.394,E2 -24391.394} C_VEL
LIN {X 0,Y 143.709,Z 527.398,A -85,B 0,C 180,E1 -24394.381,E2 -24394.381} C_VEL
LIN {X 0,Y 143.686,Z 527.401,A -85,B 0,C 180,E1 -24398.436,E2 -24398.436} C_VEL
LIN {X 0,Y 143.572,Z 527.413,A -85,B 0,C 180,E1 -24401.756,E2 -24401.756} C_VEL
LIN {X 0,Y 143.317,Z 527.444,A -85,B 0,C 180,E1 -24407.11,E2 -24407.11} C_VEL
LIN {X 0,Y 143.277,Z 527.448,A -85,B 0,C 180,E1 -24411.253,E2 -24411.253} C_VEL
LIN {X 0,Y 143.19,Z 527.461,A -85,B 0,C 180,E1 -24417.936,E2 -24417.936} C_VEL
LIN {X 0,Y 143.169,Z 527.461,A -85,B 0,C 180,E1 -24423.435,E2 -24423.435} C_VEL
LIN {X 0,Y 143.107,Z 527.471,A -85,B 0,C 180,E1 -24429.673,E2 -24429.673} C_VEL
LIN {X 0,Y 143.154,Z 527.456,A -85,B 0,C 180,E1 -24433.416,E2 -24433.416} C_VEL
LIN {X 0,Y 143.155,Z 527.465,A -85,B 0,C 180,E1 -24437.424,E2 -24437.424} C_VEL
LIN {X 0,Y 143.137,Z 527.459,A -85,B 0,C 180,E1 -24441.773,E2 -24441.773} C_VEL
LIN {X 0,Y 143.183,Z 527.46,A -85,B 0,C 180,E1 -24447.321,E2 -24447.321} C_VEL
LIN {X 0,Y 143.188,Z 527.457,A -85,B 0,C 180,E1 -24452.062,E2 -24452.062} C_VEL
LIN {X 0,Y 143.275,Z 527.448,A -85,B 0,C 180,E1 -24458.745,E2 -24458.745} C_VEL
LIN {X 0,Y 143.314,Z 527.443,A -85,B 0,C 180,E1 -24462.888,E2 -24462.888} C_VEL
LIN {X 0,Y 143.6,Z 527.403,A -85,B 0,C 180,E1 -24468.71,E2 -24468.71} C_VEL
LIN {X 0,Y 143.682,Z 527.399,A -85,B 0,C 180,E1 -24471.562,E2 -24471.562} C_VEL
LIN {X 0,Y 144.175,Z 527.329,A -85,B 0,C 180,E1 -24480,E2 -24480} C_VEL
LIN {X 0,Y 143.682,Z 527.399,A -85,B 0,C 180,E1 -24488.438,E2 -24488.438} C_VEL
LIN {X 0,Y 143.569,Z 527.413,A -85,B 0,C 180,E1 -24491.758,E2 -24491.758} C_VEL
LIN {X 0,Y 143.314,Z 527.445,A -85,B 0,C 180,E1 -24497.111,E2 -24497.111} C_VEL
LIN {X 0,Y 143.274,Z 527.452,A -85,B 0,C 180,E1 -24501.255,E2 -24501.255} C_VEL
LIN {X 0,Y 143.188,Z 527.463,A -85,B 0,C 180,E1 -24507.938,E2 -24507.938} C_VEL
LIN {X 0,Y 143.166,Z 527.466,A -85,B 0,C 180,E1 -24513.436,E2 -24513.436} C_VEL
LIN {X 0,Y 143.08,Z 527.477,A -85,B 0,C 180,E1 -24519.684,E2 -24519.684} C_VEL
LIN {X 0,Y 143.104,Z 527.475,A -85,B 0,C 180,E1 -24523.437,E2 -24523.437} C_VEL
LIN {X 0,Y 143.176,Z 527.463,A -85,B 0,C 180,E1 -24527.416,E2 -24527.416} C_VEL
LIN {X 0,Y 143.519,Z 527.447,A -85,B 0,C 180,E1 -24532.39,E2 -24532.39} C_VEL
LIN {X 0,Y 145.063,Z 532.182,A -85,B 0,C 180,E1 -24535.448,E2 -24535.448} C_VEL
LIN {X 0,Y 144.951,Z 535.755,A -85,B 0,C 180,E1 -24537.419,E2 -24537.419} C_VEL
LIN {X 0,Y 144.856,Z 536.3,A -85,B 0,C 180,E1 -24537.703,E2 -24537.703} C_VEL
LIN {X 0,Y 146.704,Z 549.038,A -85,B 0,C 180,E1 -24539.154,E2 -24539.154} C_VEL
LIN {X 0,Y 147.569,Z 558.398,A -85,B 0,C 180,E1 -24540.567,E2 -24540.567} C_VEL
LIN {X 0,Y 147.691,Z 568.121,A -85,B 0,C 180,E1 -24542.359,E2 -24542.359} C_VEL
LIN {X 0,Y 147.572,Z 576.358,A -85,B 0,C 180,E1 -24544.244,E2 -24544.244} C_VEL
LIN {X 0,Y 147.128,Z 585.664,A -85,B 0,C 180,E1 -24546.839,E2 -24546.839} C_VEL
LIN {X 0,Y 145.987,Z 591.658,A -85,B 0,C 180,E1 -24548.836,E2 -24548.836} C_VEL
LIN {X 0,Y 143.937,Z 599.924,A -85,B 0,C 180,E1 -24552.233,E2 -24552.233} C_VEL
LIN {X 0,Y 142.767,Z 605.292,A -85,B 0,C 180,E1 -24555.024,E2 -24555.024} C_VEL
LIN {X 0,Y 141.624,Z 610.7,A -85,B 0,C 180,E1 -24558.552,E2 -24558.552} C_VEL
LIN {X 0,Y 141.029,Z 614.201,A -85,B 0,C 180,E1 -24561.403,E2 -24561.403} C_VEL
LIN {X 0,Y 140.642,Z 618.178,A -85,B 0,C 180,E1 -24565.703,E2 -24565.703} C_VEL
LIN {X 0,Y 140.652,Z 619.73,A -85,B 0,C 180,E1 -24567.925,E2 -24567.925} C_VEL
LIN {X 0,Y 140.717,Z 620.866,A -85,B 0,C 180,E1 -24570.001,E2 -24570.001} C_VEL
LIN {X 0,Y 140.618,Z 621.899,A -85,B 0,C 180,E1 -24572.866,E2 -24572.866} C_VEL
LIN {X 0,Y 140.721,Z 622.462,A -85,B 0,C 180,E1 -24575.734,E2 -24575.734} C_VEL
LIN {X 0,Y 141.082,Z 622.571,A -85,B 0,C 180,E1 -24578.596,E2 -24578.596} C_VEL
LIN {X 0,Y 141.753,Z 622.189,A -85,B 0,C 180,E1 -24581.44,E2 -24581.44} C_VEL
LIN {X 0,Y 142.786,Z 621.237,A -85,B 0,C 180,E1 -24584.248,E2 -24584.248} C_VEL
LIN {X 0,Y 144.15,Z 619.809,A -85,B 0,C 180,E1 -24587.011,E2 -24587.011} C_VEL
LIN {X 0,Y 146.942,Z 616.743,A -85,B 0,C 180,E1 -24591.023,E2 -24591.023} C_VEL
LIN {X 0,Y 150.494,Z 612.41,A -85,B 0,C 180,E1 -24594.855,E2 -24594.855} C_VEL
LIN {X 0,Y 151.43,Z 611.514,A -85,B 0,C 180,E1 -24595.609,E2 -24595.609} C_VEL
LIN {X 0,Y 156.509,Z 612.442,A -85,B 0,C 180,E1 -24599.602,E2 -24599.602} C_VEL
LIN {X 0,Y 163.77,Z 612.299,A -85,B 0,C 180,E1 -24603.911,E2 -24603.911} C_VEL
LIN {X 0,Y 167.999,Z 611.728,A -85,B 0,C 180,E1 -24605.852,E2 -24605.852} C_VEL
LIN {X 0,Y 171.98,Z 610.819,A -85,B 0,C 180,E1 -24607.807,E2 -24607.807} C_VEL
LIN {X 0,Y 176.223,Z 609.406,A -85,B 0,C 180,E1 -24610.735,E2 -24610.735} C_VEL
LIN {X 0,Y 177.546,Z 608.657,A -85,B 0,C 180,E1 -24612.295,E2 -24612.295} C_VEL
LIN {X 0,Y 178.762,Z 607.695,A -85,B 0,C 180,E1 -24615.047,E2 -24615.047} C_VEL
LIN {X 0,Y 179.023,Z 607.04,A -85,B 0,C 180,E1 -24618.237,E2 -24618.237} C_VEL
LIN {X 0,Y 178.551,Z 606.811,A -85,B 0,C 180,E1 -24620.966,E2 -24620.966} C_VEL
LIN {X 0,Y 178.192,Z 606.814,A -85,B 0,C 180,E1 -24622.076,E2 -24622.076} C_VEL
LIN {X 0,Y 177.05,Z 606.904,A -85,B 0,C 180,E1 -24623.457,E2 -24623.457} C_VEL
LIN {X 0,Y 172.841,Z 607.378,A -85,B 0,C 180,E1 -24625.235,E2 -24625.235} C_VEL
LIN {X 0,Y 170.236,Z 607.591,A -85,B 0,C 180,E1 -24626.219,E2 -24626.219} C_VEL
LIN {X 0,Y 164.1,Z 607.707,A -85,B 0,C 180,E1 -24627.936,E2 -24627.936} C_VEL
LIN {X 0,Y 154.634,Z 606.729,A -85,B 0,C 180,E1 -24630.52,E2 -24630.52} C_VEL
LIN {X 0,Y 150.782,Z 605.761,A -85,B 0,C 180,E1 -24632.153,E2 -24632.153} C_VEL
LIN {X 0,Y 149.78,Z 605.333,A -85,B 0,C 180,E1 -24632.778,E2 -24632.778} C_VEL
LIN {X 0,Y 143.177,Z 601.192,A -85,B 0,C 180,E1 -24638.399,E2 -24638.399} C_VEL
LIN {X 0,Y 139.727,Z 597.367,A -85,B 0,C 180,E1 -24642.435,E2 -24642.435} C_VEL
LIN {X 0,Y 136.987,Z 590.932,A -85,B 0,C 180,E1 -24648.158,E2 -24648.158} C_VEL
LIN {X 0,Y 136.091,Z 584.811,A -85,B 0,C 180,E1 -24652.582,E2 -24652.582} C_VEL
LIN {X 0,Y 135.713,Z 577.219,A -85,B 0,C 180,E1 -24657.032,E2 -24657.032} C_VEL
LIN {X 0,Y 135.678,Z 576.534,A -85,B 0,C 180,E1 -24657.495,E2 -24657.495} C_VEL
LIN {X 0,Y 135.347,Z 577.836,A -85,B 0,C 180,E1 -24658.513,E2 -24658.513} C_VEL
LIN {X 0,Y 138.242,Z 578.885,A -85,B 0,C 180,E1 -24662.914,E2 -24662.914} C_VEL
LIN {X 0,Y 144.448,Z 579.083,A -85,B 0,C 180,E1 -24668.393,E2 -24668.393} C_VEL
LIN {X 0,Y 147.66,Z 579.751,A -85,B 0,C 180,E1 -24670.975,E2 -24670.975} C_VEL
LIN {X 0,Y 156.406,Z 579.437,A -85,B 0,C 180,E1 -24675.641,E2 -24675.641} C_VEL
LIN {X 0,Y 158.232,Z 580.018,A -85,B 0,C 180,E1 -24676.781,E2 -24676.781} C_VEL
LIN {X 0,Y 158.596,Z 580.916,A -85,B 0,C 180,E1 -24677.405,E2 -24677.405} C_VEL
LIN {X 0,Y 157.252,Z 587.368,A -85,B 0,C 180,E1 -24680.188,E2 -24680.188} C_VEL
LIN {X 0,Y 156.081,Z 591.02,A -85,B 0,C 180,E1 -24681.814,E2 -24681.814} C_VEL
LIN {X 0,Y 151.969,Z 597.588,A -85,B 0,C 180,E1 -24684.596,E2 -24684.596} C_VEL
LIN {X 0,Y 147.845,Z 603.11,A -85,B 0,C 180,E1 -24687.682,E2 -24687.682} C_VEL
LIN {X 0,Y 145.579,Z 605.955,A -85,B 0,C 180,E1 -24689.658,E2 -24689.658} C_VEL
LIN {X 0,Y 142.379,Z 609.607,A -85,B 0,C 180,E1 -24692.948,E2 -24692.948} C_VEL
LIN {X 0,Y 138.9,Z 612.907,A -85,B 0,C 180,E1 -24697.386,E2 -24697.386} C_VEL
LIN {X 0,Y 137.39,Z 614.208,A -85,B 0,C 180,E1 -24699.885,E2 -24699.885} C_VEL
LIN {X 0,Y 135.611,Z 615.304,A -85,B 0,C 180,E1 -24703.484,E2 -24703.484} C_VEL
LIN {X 0,Y 134.337,Z 615.643,A -85,B 0,C 180,E1 -24707.146,E2 -24707.146} C_VEL
LIN {X 0,Y 133.261,Z 614.816,A -85,B 0,C 180,E1 -24712.287,E2 -24712.287} C_VEL
LIN {X 0,Y 133.062,Z 614.099,A -85,B 0,C 180,E1 -24714.478,E2 -24714.478} C_VEL
LIN {X 0,Y 133.09,Z 612.226,A -85,B 0,C 180,E1 -24718.124,E2 -24718.124} C_VEL
LIN {X 0,Y 133.835,Z 608.228,A -85,B 0,C 180,E1 -24723.216,E2 -24723.216} C_VEL
LIN {X 0,Y 134.718,Z 604.123,A -85,B 0,C 180,E1 -24726.965,E2 -24726.965} C_VEL
LIN {X 0,Y 135.842,Z 599.403,A -85,B 0,C 180,E1 -24730.348,E2 -24730.348} C_VEL
LIN {X 0,Y 137.215,Z 593.669,A -85,B 0,C 180,E1 -24733.638,E2 -24733.638} C_VEL
LIN {X 0,Y 139.108,Z 586.619,A -85,B 0,C 180,E1 -24736.857,E2 -24736.857} C_VEL
LIN {X 0,Y 141.273,Z 577.913,A -85,B 0,C 180,E1 -24739.971,E2 -24739.971} C_VEL
LIN {X 0,Y 142.017,Z 574.041,A -85,B 0,C 180,E1 -24741.102,E2 -24741.102} C_VEL
LIN {X 0,Y 141.667,Z 563.887,A -85,B 0,C 180,E1 -24743.947,E2 -24743.947} C_VEL
LIN {X 0,Y 140.632,Z 553.068,A -85,B 0,C 180,E1 -24746.345,E2 -24746.345} C_VEL
LIN {X 0,Y 139.109,Z 542.944,A -85,B 0,C 180,E1 -24748.189,E2 -24748.189} C_VEL
LIN {X 0,Y 137.089,Z 533.016,A -85,B 0,C 180,E1 -24749.723,E2 -24749.723} C_VEL
LIN {X 0,Y 137.352,Z 531.338,A -85,B 0,C 180,E1 -24751.465,E2 -24751.465} C_VEL
LIN {X 0,Y 136.624,Z 528.28,A -85,B 0,C 180,E1 -24755.163,E2 -24755.163} C_VEL
LIN {X 0,Y 136.61,Z 528.282,A -85,B 0,C 180,E1 -24758.877,E2 -24758.877} C_VEL
LIN {X 0,Y 136.494,Z 528.295,A -85,B 0,C 180,E1 -24761.956,E2 -24761.956} C_VEL
LIN {X 0,Y 136.253,Z 528.325,A -85,B 0,C 180,E1 -24768.027,E2 -24768.027} C_VEL
LIN {X 0,Y 136.198,Z 528.331,A -85,B 0,C 180,E1 -24771.747,E2 -24771.747} C_VEL
LIN {X 0,Y 136.116,Z 528.342,A -85,B 0,C 180,E1 -24778.627,E2 -24778.627} C_VEL
LIN {X 0,Y 136.08,Z 528.341,A -85,B 0,C 180,E1 -24784.616,E2 -24784.616} C_VEL
LIN {X 0,Y 136.076,Z 528.346,A -85,B 0,C 180,E1 -24789.22,E2 -24789.22} C_VEL
LIN {X 0,Y 136.091,Z 528.337,A -85,B 0,C 180,E1 -24793.698,E2 -24793.698} C_VEL
LIN {X 0,Y 136.104,Z 528.344,A -85,B 0,C 180,E1 -24797.834,E2 -24797.834} C_VEL
LIN {X 0,Y 136.089,Z 528.337,A -85,B 0,C 180,E1 -24801.705,E2 -24801.705} C_VEL
LIN {X 0,Y 136.09,Z 528.34,A -85,B 0,C 180,E1 -24805.716,E2 -24805.716} C_VEL
LIN {X 0,Y 136.144,Z 528.333,A -85,B 0,C 180,E1 -24812.316,E2 -24812.316} C_VEL
LIN {X 0,Y 136.242,Z 528.324,A -85,B 0,C 180,E1 -24818.832,E2 -24818.832} C_VEL
LIN {X 0,Y 136.283,Z 528.321,A -85,B 0,C 180,E1 -24825.058,E2 -24825.058} C_VEL
LIN {X 0,Y 136.499,Z 528.289,A -85,B 0,C 180,E1 -24828.115,E2 -24828.115} C_VEL
LIN {X 0,Y 136.606,Z 528.279,A -85,B 0,C 180,E1 -24831.121,E2 -24831.121} C_VEL
LIN {X 0,Y 137.132,Z 528.205,A -85,B 0,C 180,E1 -24840,E2 -24840} C_VEL
LIN {X 0,Y 136.606,Z 528.28,A -85,B 0,C 180,E1 -24848.878,E2 -24848.878} C_VEL
LIN {X 0,Y 136.49,Z 528.295,A -85,B 0,C 180,E1 -24851.958,E2 -24851.958} C_VEL
LIN {X 0,Y 136.249,Z 528.328,A -85,B 0,C 180,E1 -24858.028,E2 -24858.028} C_VEL
LIN {X 0,Y 136.195,Z 528.335,A -85,B 0,C 180,E1 -24861.749,E2 -24861.749} C_VEL
LIN {X 0,Y 136.098,Z 528.345,A -85,B 0,C 180,E1 -24868.617,E2 -24868.617} C_VEL
LIN {X 0,Y 136.076,Z 528.346,A -85,B 0,C 180,E1 -24874.619,E2 -24874.619} C_VEL
LIN {X 0,Y 136.054,Z 528.35,A -85,B 0,C 180,E1 -24879.212,E2 -24879.212} C_VEL
LIN {X 0,Y 136.046,Z 528.353,A -85,B 0,C 180,E1 -24883.681,E2 -24883.681} C_VEL
LIN {X 0,Y 136.359,Z 528.313,A -85,B 0,C 180,E1 -24891.076,E2 -24891.076} C_VEL
LIN {X 0,Y 138.236,Z 534.046,A -85,B 0,C 180,E1 -24895.207,E2 -24895.207} C_VEL
LIN {X 0,Y 138.187,Z 536.522,A -85,B 0,C 180,E1 -24896.551,E2 -24896.551} C_VEL
LIN {X 0,Y 139.982,Z 548.927,A -85,B 0,C 180,E1 -24898.065,E2 -24898.065} C_VEL
LIN {X 0,Y 140.83,Z 559.01,A -85,B 0,C 180,E1 -24899.683,E2 -24899.683} C_VEL
LIN {X 0,Y 140.914,Z 567.422,A -85,B 0,C 180,E1 -24901.314,E2 -24901.314} C_VEL
LIN {X 0,Y 140.743,Z 575.789,A -85,B 0,C 180,E1 -24903.296,E2 -24903.296} C_VEL
LIN {X 0,Y 140.293,Z 584.368,A -85,B 0,C 180,E1 -24905.769,E2 -24905.769} C_VEL
LIN {X 0,Y 139.827,Z 588.247,A -85,B 0,C 180,E1 -24907.076,E2 -24907.076} C_VEL
LIN {X 0,Y 138.425,Z 593.94,A -85,B 0,C 180,E1 -24909.184,E2 -24909.184} C_VEL
LIN {X 0,Y 136.799,Z 600.267,A -85,B 0,C 180,E1 -24912.048,E2 -24912.048} C_VEL
LIN {X 0,Y 135.616,Z 605.539,A -85,B 0,C 180,E1 -24914.984,E2 -24914.984} C_VEL
LIN {X 0,Y 134.667,Z 609.914,A -85,B 0,C 180,E1 -24917.952,E2 -24917.952} C_VEL
LIN {X 0,Y 133.812,Z 615.031,A -85,B 0,C 180,E1 -24922.457,E2 -24922.457} C_VEL
LIN {X 0,Y 133.567,Z 618.747,A -85,B 0,C 180,E1 -24926.985,E2 -24926.985} C_VEL
LIN {X 0,Y 133.559,Z 620.98,A -85,B 0,C 180,E1 -24931.168,E2 -24931.168} C_VEL
LIN {X 0,Y 133.652,Z 622.217,A -85,B 0,C 180,E1 -24936.038,E2 -24936.038} C_VEL
LIN {X 0,Y 134.068,Z 622.421,A -85,B 0,C 180,E1 -24939.05,E2 -24939.05} C_VEL
LIN {X 0,Y 134.796,Z 622.059,A -85,B 0,C 180,E1 -24942.039,E2 -24942.039} C_VEL
LIN {X 0,Y 135.908,Z 621.2,A -85,B 0,C 180,E1 -24944.986,E2 -24944.986} C_VEL
LIN {X 0,Y 137.382,Z 619.885,A -85,B 0,C 180,E1 -24947.876,E2 -24947.876} C_VEL
LIN {X 0,Y 140.348,Z 616.946,A -85,B 0,C 180,E1 -24952.061,E2 -24952.061} C_VEL
LIN {X 0,Y 144.097,Z 612.784,A -85,B 0,C 180,E1 -24956.039,E2 -24956.039} C_VEL
LIN {X 0,Y 146.235,Z 610.541,A -85,B 0,C 180,E1 -24957.749,E2 -24957.749} C_VEL
LIN {X 0,Y 154.003,Z 611.888,A -85,B 0,C 180,E1 -24963.206,E2 -24963.206} C_VEL
LIN {X 0,Y 162.3,Z 611.587,A -85,B 0,C 180,E1 -24967.319,E2 -24967.319} C_VEL
LIN {X 0,Y 166.319,Z 611.003,A -85,B 0,C 180,E1 -24969.336,E2 -24969.336} C_VEL
LIN {X 0,Y 169.853,Z 610.017,A -85,B 0,C 180,E1 -24971.86,E2 -24971.86} C_VEL
LIN {X 0,Y 171.297,Z 609.281,A -85,B 0,C 180,E1 -24974.226,E2 -24974.226} C_VEL
LIN {X 0,Y 171.808,Z 608.84,A -85,B 0,C 180,E1 -24975.941,E2 -24975.941} C_VEL
LIN {X 0,Y 171.837,Z 608.275,A -85,B 0,C 180,E1 -24979.127,E2 -24979.127} C_VEL
LIN {X 0,Y 171.449,Z 608.031,A -85,B 0,C 180,E1 -24981.157,E2 -24981.157} C_VEL
LIN {X 0,Y 171.03,Z 607.998,A -85,B 0,C 180,E1 -24981.948,E2 -24981.948} C_VEL
LIN {X 0,Y 166.975,Z 608.158,A -85,B 0,C 180,E1 -24983.896,E2 -24983.896} C_VEL
LIN {X 0,Y 162.447,Z 608.132,A -85,B 0,C 180,E1 -24985.777,E2 -24985.777} C_VEL
LIN {X 0,Y 154.226,Z 606.836,A -85,B 0,C 180,E1 -24989.917,E2 -24989.917} C_VEL
LIN {X 0,Y 149.78,Z 605.333,A -85,B 0,C 180,E1 -24992.778,E2 -24992.778} C_VEL
LIN {X 0,Y 146.581,Z 604.014,A -85,B 0,C 180,E1 -24994.619,E2 -24994.619} C_VEL
LIN {X 0,Y 140.26,Z 601.011,A -85,B 0,C 180,E1 -24997.434,E2 -24997.434} C_VEL
LIN {X 0,Y 134.588,Z 597.234,A -85,B 0,C 180,E1 -25000.453,E2 -25000.453} C_VEL
LIN {X 0,Y 132.504,Z 594.714,A -85,B 0,C 180,E1 -25002.578,E2 -25002.578} C_VEL
LIN {X 0,Y 130.798,Z 590.537,A -85,B 0,C 180,E1 -25006.2,E2 -25006.2} C_VEL
LIN {X 0,Y 129.665,Z 584.654,A -85,B 0,C 180,E1 -25010.642,E2 -25010.642} C_VEL
LIN {X 0,Y 129.299,Z 581.537,A -85,B 0,C 180,E1 -25012.779,E2 -25012.779} C_VEL
LIN {X 0,Y 128.829,Z 582.546,A -85,B 0,C 180,E1 -25013.736,E2 -25013.736} C_VEL
LIN {X 0,Y 130.08,Z 582.967,A -85,B 0,C 180,E1 -25016.903,E2 -25016.903} C_VEL
LIN {X 0,Y 133.764,Z 584.295,A -85,B 0,C 180,E1 -25023.354,E2 -25023.354} C_VEL
LIN {X 0,Y 139.622,Z 584.447,A -85,B 0,C 180,E1 -25028.686,E2 -25028.686} C_VEL
LIN {X 0,Y 143.676,Z 585.082,A -85,B 0,C 180,E1 -25031.948,E2 -25031.948} C_VEL
LIN {X 0,Y 151.489,Z 584.828,A -85,B 0,C 180,E1 -25036.162,E2 -25036.162} C_VEL
LIN {X 0,Y 152.321,Z 586.421,A -85,B 0,C 180,E1 -25037.452,E2 -25037.452} C_VEL
LIN {X 0,Y 150.087,Z 592.845,A -85,B 0,C 180,E1 -25040.521,E2 -25040.521} C_VEL
LIN {X 0,Y 145.57,Z 599.198,A -85,B 0,C 180,E1 -25043.462,E2 -25043.462} C_VEL
LIN {X 0,Y 141.381,Z 604.324,A -85,B 0,C 180,E1 -25046.576,E2 -25046.576} C_VEL
LIN {X 0,Y 137.766,Z 608.335,A -85,B 0,C 180,E1 -25049.858,E2 -25049.858} C_VEL
LIN {X 0,Y 134.586,Z 611.431,A -85,B 0,C 180,E1 -25053.328,E2 -25053.328} C_VEL
LIN {X 0,Y 131.862,Z 613.651,A -85,B 0,C 180,E1 -25056.918,E2 -25056.918} C_VEL
LIN {X 0,Y 129.708,Z 615.072,A -85,B 0,C 180,E1 -25060.66,E2 -25060.66} C_VEL
LIN {X 0,Y 127.593,Z 615.828,A -85,B 0,C 180,E1 -25065.731,E2 -25065.731} C_VEL
LIN {X 0,Y 126.314,Z 615.132,A -85,B 0,C 180,E1 -25071.165,E2 -25071.165} C_VEL
LIN {X 0,Y 125.949,Z 612.875,A -85,B 0,C 180,E1 -25076.826,E2 -25076.826} C_VEL
LIN {X 0,Y 126.386,Z 609.876,A -85,B 0,C 180,E1 -25081.403,E2 -25081.403} C_VEL
LIN {X 0,Y 127.442,Z 605.067,A -85,B 0,C 180,E1 -25086.432,E2 -25086.432} C_VEL
LIN {X 0,Y 128.477,Z 600.712,A -85,B 0,C 180,E1 -25089.875,E2 -25089.875} C_VEL
LIN {X 0,Y 129.912,Z 594.936,A -85,B 0,C 180,E1 -25093.498,E2 -25093.498} C_VEL
LIN {X 0,Y 131.326,Z 589.764,A -85,B 0,C 180,E1 -25096.153,E2 -25096.153} C_VEL
LIN {X 0,Y 133.158,Z 583.037,A -85,B 0,C 180,E1 -25098.968,E2 -25098.968} C_VEL
LIN {X 0,Y 135.023,Z 575.615,A -85,B 0,C 180,E1 -25101.478,E2 -25101.478} C_VEL
LIN {X 0,Y 135.021,Z 569.215,A -85,B 0,C 180,E1 -25103.473,E2 -25103.473} C_VEL
LIN {X 0,Y 134.609,Z 561.729,A -85,B 0,C 180,E1 -25105.507,E2 -25105.507} C_VEL
LIN {X 0,Y 133.868,Z 553.571,A -85,B 0,C 180,E1 -25107.396,E2 -25107.396} C_VEL
LIN {X 0,Y 132.494,Z 544,A -85,B 0,C 180,E1 -25109.267,E2 -25109.267} C_VEL
LIN {X 0,Y 130.675,Z 535.172,A -85,B 0,C 180,E1 -25110.721,E2 -25110.721} C_VEL
LIN {X 0,Y 130.277,Z 533.046,A -85,B 0,C 180,E1 -25111.158,E2 -25111.158} C_VEL
LIN {X 0,Y 130.141,Z 531.374,A -85,B 0,C 180,E1 -25113.094,E2 -25113.094} C_VEL
LIN {X 0,Y 129.557,Z 529.16,A -85,B 0,C 180,E1 -25115.836,E2 -25115.836} C_VEL
LIN {X 0,Y 129.532,Z 529.163,A -85,B 0,C 180,E1 -25119.366,E2 -25119.366} C_VEL
LIN {X 0,Y 129.395,Z 529.18,A -85,B 0,C 180,E1 -25122.546,E2 -25122.546} C_VEL
LIN {X 0,Y 129.16,Z 529.204,A -85,B 0,C 180,E1 -25129.053,E2 -25129.053} C_VEL
LIN {X 0,Y 129.108,Z 529.211,A -85,B 0,C 180,E1 -25132.397,E2 -25132.397} C_VEL
LIN {X 0,Y 129.035,Z 529.223,A -85,B 0,C 180,E1 -25139.372,E2 -25139.372} C_VEL
LIN {X 0,Y 128.996,Z 529.223,A -85,B 0,C 180,E1 -25145.191,E2 -25145.191} C_VEL
LIN {X 0,Y 129.006,Z 529.223,A -85,B 0,C 180,E1 -25150.822,E2 -25150.822} C_VEL
LIN {X 0,Y 129.023,Z 529.222,A -85,B 0,C 180,E1 -25155.08,E2 -25155.08} C_VEL
LIN {X 0,Y 129.013,Z 529.226,A -85,B 0,C 180,E1 -25159.696,E2 -25159.696} C_VEL
LIN {X 0,Y 129.022,Z 529.219,A -85,B 0,C 180,E1 -25164.79,E2 -25164.79} C_VEL
LIN {X 0,Y 129.049,Z 529.221,A -85,B 0,C 180,E1 -25170.65,E2 -25170.65} C_VEL
LIN {X 0,Y 129.105,Z 529.216,A -85,B 0,C 180,E1 -25177.727,E2 -25177.727} C_VEL
LIN {X 0,Y 129.157,Z 529.202,A -85,B 0,C 180,E1 -25180.944,E2 -25180.944} C_VEL
LIN {X 0,Y 129.416,Z 529.173,A -85,B 0,C 180,E1 -25187.815,E2 -25187.815} C_VEL
LIN {X 0,Y 129.528,Z 529.161,A -85,B 0,C 180,E1 -25190.632,E2 -25190.632} C_VEL
LIN {X 0,Y 130.088,Z 529.082,A -85,B 0,C 180,E1 -25200,E2 -25200} C_VEL
LIN {X 0,Y 129.528,Z 529.163,A -85,B 0,C 180,E1 -25209.368,E2 -25209.368} C_VEL
LIN {X 0,Y 129.392,Z 529.179,A -85,B 0,C 180,E1 -25212.548,E2 -25212.548} C_VEL
LIN {X 0,Y 129.157,Z 529.211,A -85,B 0,C 180,E1 -25219.055,E2 -25219.055} C_VEL
LIN {X 0,Y 129.106,Z 529.218,A -85,B 0,C 180,E1 -25222.399,E2 -25222.399} C_VEL
LIN {X 0,Y 129.033,Z 529.227,A -85,B 0,C 180,E1 -25229.374,E2 -25229.374} C_VEL
LIN {X 0,Y 128.991,Z 529.23,A -85,B 0,C 180,E1 -25235.191,E2 -25235.191} C_VEL
LIN {X 0,Y 128.985,Z 529.231,A -85,B 0,C 180,E1 -25240.832,E2 -25240.832} C_VEL
LIN {X 0,Y 129.011,Z 529.227,A -85,B 0,C 180,E1 -25245.087,E2 -25245.087} C_VEL
LIN {X 0,Y 129.251,Z 529.397,A -85,B 0,C 180,E1 -25250.178,E2 -25250.178} C_VEL
LIN {X 0,Y 131.412,Z 536.275,A -85,B 0,C 180,E1 -25255.214,E2 -25255.214} C_VEL
LIN {X 0,Y 133.23,Z 548.603,A -85,B 0,C 180,E1 -25256.822,E2 -25256.822} C_VEL
LIN {X 0,Y 134.062,Z 559.047,A -85,B 0,C 180,E1 -25258.602,E2 -25258.602} C_VEL
LIN {X 0,Y 134.171,Z 566.648,A -85,B 0,C 180,E1 -25260.159,E2 -25260.159} C_VEL
LIN {X 0,Y 133.949,Z 575.355,A -85,B 0,C 180,E1 -25262.311,E2 -25262.311} C_VEL
LIN {X 0,Y 133.391,Z 584.481,A -85,B 0,C 180,E1 -25265.072,E2 -25265.072} C_VEL
LIN {X 0,Y 132.525,Z 589.761,A -85,B 0,C 180,E1 -25266.978,E2 -25266.978} C_VEL
LIN {X 0,Y 130.444,Z 597.674,A -85,B 0,C 180,E1 -25270.324,E2 -25270.324} C_VEL
LIN {X 0,Y 128.737,Z 604.594,A -85,B 0,C 180,E1 -25274.161,E2 -25274.161} C_VEL
LIN {X 0,Y 127.7,Z 609.106,A -85,B 0,C 180,E1 -25277.284,E2 -25277.284} C_VEL
LIN {X 0,Y 127.007,Z 612.84,A -85,B 0,C 180,E1 -25280.446,E2 -25280.446} C_VEL
LIN {X 0,Y 126.514,Z 617.058,A -85,B 0,C 180,E1 -25285.222,E2 -25285.222} C_VEL
LIN {X 0,Y 126.547,Z 619.962,A -85,B 0,C 180,E1 -25290.002,E2 -25290.002} C_VEL
LIN {X 0,Y 126.448,Z 621.204,A -85,B 0,C 180,E1 -25293.188,E2 -25293.188} C_VEL
LIN {X 0,Y 126.583,Z 621.971,A -85,B 0,C 180,E1 -25296.377,E2 -25296.377} C_VEL
LIN {X 0,Y 127.053,Z 622.222,A -85,B 0,C 180,E1 -25299.554,E2 -25299.554} C_VEL
LIN {X 0,Y 127.865,Z 621.922,A -85,B 0,C 180,E1 -25302.702,E2 -25302.702} C_VEL
LIN {X 0,Y 129.064,Z 621.175,A -85,B 0,C 180,E1 -25305.801,E2 -25305.801} C_VEL
LIN {X 0,Y 130.652,Z 619.975,A -85,B 0,C 180,E1 -25308.831,E2 -25308.831} C_VEL
LIN {X 0,Y 133.787,Z 617.154,A -85,B 0,C 180,E1 -25313.204,E2 -25313.204} C_VEL
LIN {X 0,Y 137.769,Z 613.118,A -85,B 0,C 180,E1 -25317.332,E2 -25317.332} C_VEL
LIN {X 0,Y 141.319,Z 609.549,A -85,B 0,C 180,E1 -25320.03,E2 -25320.03} C_VEL
LIN {X 0,Y 144.455,Z 610.42,A -85,B 0,C 180,E1 -25322.357,E2 -25322.357} C_VEL
LIN {X 0,Y 152.227,Z 611.284,A -85,B 0,C 180,E1 -25326.885,E2 -25326.885} C_VEL
LIN {X 0,Y 156.711,Z 611.238,A -85,B 0,C 180,E1 -25328.894,E2 -25328.894} C_VEL
LIN {X 0,Y 160.737,Z 610.872,A -85,B 0,C 180,E1 -25330.986,E2 -25330.986} C_VEL
LIN {X 0,Y 163.287,Z 610.363,A -85,B 0,C 180,E1 -25332.972,E2 -25332.972} C_VEL
LIN {X 0,Y 164.834,Z 609.497,A -85,B 0,C 180,E1 -25336.985,E2 -25336.985} C_VEL
LIN {X 0,Y 164.539,Z 608.913,A -85,B 0,C 180,E1 -25340.252,E2 -25340.252} C_VEL
LIN {X 0,Y 161.293,Z 608.736,A -85,B 0,C 180,E1 -25342.409,E2 -25342.409} C_VEL
LIN {X 0,Y 152.207,Z 607.666,A -85,B 0,C 180,E1 -25346.352,E2 -25346.352} C_VEL
LIN {X 0,Y 144.415,Z 605.115,A -85,B 0,C 180,E1 -25350.879,E2 -25350.879} C_VEL
LIN {X 0,Y 139.477,Z 602.35,A -85,B 0,C 180,E1 -25354.641,E2 -25354.641} C_VEL
LIN {X 0,Y 135.434,Z 598.716,A -85,B 0,C 180,E1 -25358.701,E2 -25358.701} C_VEL
LIN {X 0,Y 132.504,Z 594.714,A -85,B 0,C 180,E1 -25362.578,E2 -25362.578} C_VEL
LIN {X 0,Y 130.959,Z 592.915,A -85,B 0,C 180,E1 -25364.054,E2 -25364.054} C_VEL
LIN {X 0,Y 125.4,Z 589.152,A -85,B 0,C 180,E1 -25367.199,E2 -25367.199} C_VEL
LIN {X 0,Y 123.401,Z 587.978,A -85,B 0,C 180,E1 -25369.048,E2 -25369.048} C_VEL
LIN {X 0,Y 123.088,Z 587.674,A -85,B 0,C 180,E1 -25370.532,E2 -25370.532} C_VEL
LIN {X 0,Y 124.021,Z 587.708,A -85,B 0,C 180,E1 -25373.493,E2 -25373.493} C_VEL
LIN {X 0,Y 128.451,Z 589.281,A -85,B 0,C 180,E1 -25383.137,E2 -25383.137} C_VEL
LIN {X 0,Y 135.579,Z 589.582,A -85,B 0,C 180,E1 -25389.96,E2 -25389.96} C_VEL
LIN {X 0,Y 137.734,Z 589.879,A -85,B 0,C 180,E1 -25391.777,E2 -25391.777} C_VEL
LIN {X 0,Y 146.157,Z 589.956,A -85,B 0,C 180,E1 -25396.769,E2 -25396.769} C_VEL
LIN {X 0,Y 144.447,Z 594.078,A -85,B 0,C 180,E1 -25398.896,E2 -25398.896} C_VEL
LIN {X 0,Y 139.972,Z 599.951,A -85,B 0,C 180,E1 -25401.734,E2 -25401.734} C_VEL
LIN {X 0,Y 136.279,Z 604.201,A -85,B 0,C 180,E1 -25404.366,E2 -25404.366} C_VEL
LIN {X 0,Y 132.194,Z 608.381,A -85,B 0,C 180,E1 -25407.804,E2 -25407.804} C_VEL
LIN {X 0,Y 128.295,Z 611.879,A -85,B 0,C 180,E1 -25411.887,E2 -25411.887} C_VEL
LIN {X 0,Y 126.774,Z 613.076,A -85,B 0,C 180,E1 -25413.738,E2 -25413.738} C_VEL
LIN {X 0,Y 123.41,Z 615.16,A -85,B 0,C 180,E1 -25418.788,E2 -25418.788} C_VEL
LIN {X 0,Y 122.032,Z 615.791,A -85,B 0,C 180,E1 -25421.52,E2 -25421.52} C_VEL
LIN {X 0,Y 120.494,Z 616.016,A -85,B 0,C 180,E1 -25425.577,E2 -25425.577} C_VEL
LIN {X 0,Y 119.412,Z 615.434,A -85,B 0,C 180,E1 -25429.918,E2 -25429.918} C_VEL
LIN {X 0,Y 118.932,Z 614.259,A -85,B 0,C 180,E1 -25433.775,E2 -25433.775} C_VEL
LIN {X 0,Y 118.893,Z 612.277,A -85,B 0,C 180,E1 -25437.857,E2 -25437.857} C_VEL
LIN {X 0,Y 119.384,Z 609.432,A -85,B 0,C 180,E1 -25442.011,E2 -25442.011} C_VEL
LIN {X 0,Y 120.154,Z 605.979,A -85,B 0,C 180,E1 -25445.828,E2 -25445.828} C_VEL
LIN {X 0,Y 121.556,Z 600.267,A -85,B 0,C 180,E1 -25450.581,E2 -25450.581} C_VEL
LIN {X 0,Y 123.126,Z 594.295,A -85,B 0,C 180,E1 -25454.441,E2 -25454.441} C_VEL
LIN {X 0,Y 125.006,Z 587.685,A -85,B 0,C 180,E1 -25457.827,E2 -25457.827} C_VEL
LIN {X 0,Y 127.361,Z 579.185,A -85,B 0,C 180,E1 -25461.265,E2 -25461.265} C_VEL
LIN {X 0,Y 128.266,Z 575.313,A -85,B 0,C 180,E1 -25462.52,E2 -25462.52} C_VEL
LIN {X 0,Y 128.132,Z 566.699,A -85,B 0,C 180,E1 -25465.279,E2 -25465.279} C_VEL
LIN {X 0,Y 127.371,Z 555.888,A -85,B 0,C 180,E1 -25468.141,E2 -25468.141} C_VEL
LIN {X 0,Y 126.019,Z 545.723,A -85,B 0,C 180,E1 -25470.298,E2 -25470.298} C_VEL
LIN {X 0,Y 124.226,Z 536.741,A -85,B 0,C 180,E1 -25471.923,E2 -25471.923} C_VEL
LIN {X 0,Y 123.249,Z 533.301,A -85,B 0,C 180,E1 -25472.552,E2 -25472.552} C_VEL
LIN {X 0,Y 122.446,Z 530.046,A -85,B 0,C 180,E1 -25476.797,E2 -25476.797} C_VEL
LIN {X 0,Y 122.458,Z 530.044,A -85,B 0,C 180,E1 -25479.912,E2 -25479.912} C_VEL
LIN {X 0,Y 122.265,Z 530.067,A -85,B 0,C 180,E1 -25483.291,E2 -25483.291} C_VEL
LIN {X 0,Y 122.05,Z 530.092,A -85,B 0,C 180,E1 -25490.21,E2 -25490.21} C_VEL
LIN {X 0,Y 121.983,Z 530.098,A -85,B 0,C 180,E1 -25493.783,E2 -25493.783} C_VEL
LIN {X 0,Y 121.941,Z 530.108,A -85,B 0,C 180,E1 -25500.172,E2 -25500.172} C_VEL
LIN {X 0,Y 121.922,Z 530.107,A -85,B 0,C 180,E1 -25506.195,E2 -25506.195} C_VEL
LIN {X 0,Y 121.936,Z 530.102,A -85,B 0,C 180,E1 -25511.472,E2 -25511.472} C_VEL
LIN {X 0,Y 121.941,Z 530.107,A -85,B 0,C 180,E1 -25518.523,E2 -25518.523} C_VEL
LIN {X 0,Y 121.974,Z 530.096,A -85,B 0,C 180,E1 -25524.817,E2 -25524.817} C_VEL
LIN {X 0,Y 121.94,Z 530.109,A -85,B 0,C 180,E1 -25529.825,E2 -25529.825} C_VEL
LIN {X 0,Y 121.981,Z 530.104,A -85,B 0,C 180,E1 -25536.215,E2 -25536.215} C_VEL
LIN {X 0,Y 122.047,Z 530.091,A -85,B 0,C 180,E1 -25539.787,E2 -25539.787} C_VEL
LIN {X 0,Y 122.262,Z 530.066,A -85,B 0,C 180,E1 -25546.707,E2 -25546.707} C_VEL
LIN {X 0,Y 122.454,Z 530.04,A -85,B 0,C 180,E1 -25550.085,E2 -25550.085} C_VEL
LIN {X 0,Y 122.608,Z 530.018,A -85,B 0,C 180,E1 -25556.714,E2 -25556.714} C_VEL
LIN {X 0,Y 123.042,Z 529.959,A -85,B 0,C 180,E1 -25560,E2 -25560} C_VEL
LIN {X 0,Y 122.454,Z 530.041,A -85,B 0,C 180,E1 -25566.591,E2 -25566.591} C_VEL
LIN {X 0,Y 122.454,Z 530.045,A -85,B 0,C 180,E1 -25569.914,E2 -25569.914} C_VEL
LIN {X 0,Y 122.262,Z 530.068,A -85,B 0,C 180,E1 -25573.293,E2 -25573.293} C_VEL
LIN {X 0,Y 122.046,Z 530.096,A -85,B 0,C 180,E1 -25580.213,E2 -25580.213} C_VEL
LIN {X 0,Y 121.981,Z 530.106,A -85,B 0,C 180,E1 -25583.785,E2 -25583.785} C_VEL
LIN {X 0,Y 121.939,Z 530.11,A -85,B 0,C 180,E1 -25590.174,E2 -25590.174} C_VEL
LIN {X 0,Y 121.911,Z 530.111,A -85,B 0,C 180,E1 -25596.191,E2 -25596.191} C_VEL
LIN {X 0,Y 121.919,Z 530.11,A -85,B 0,C 180,E1 -25601.466,E2 -25601.466} C_VEL
LIN {X 0,Y 122.052,Z 530.104,A -85,B 0,C 180,E1 -25608.735,E2 -25608.735} C_VEL
LIN {X 0,Y 124.007,Z 536.215,A -85,B 0,C 180,E1 -25613.636,E2 -25613.636} C_VEL
LIN {X 0,Y 125.405,Z 539.824,A -85,B 0,C 180,E1 -25614.28,E2 -25614.28} C_VEL
LIN {X 0,Y 126.722,Z 550.29,A -85,B 0,C 180,E1 -25615.821,E2 -25615.821} C_VEL
LIN {X 0,Y 127.446,Z 561.04,A -85,B 0,C 180,E1 -25617.823,E2 -25617.823} C_VEL
LIN {X 0,Y 127.265,Z 572.53,A -85,B 0,C 180,E1 -25620.542,E2 -25620.542} C_VEL
LIN {X 0,Y 126.726,Z 581.414,A -85,B 0,C 180,E1 -25623.222,E2 -25623.222} C_VEL
LIN {X 0,Y 125.98,Z 588.276,A -85,B 0,C 180,E1 -25625.707,E2 -25625.707} C_VEL
LIN {X 0,Y 124.249,Z 594.739,A -85,B 0,C 180,E1 -25628.43,E2 -25628.43} C_VEL
LIN {X 0,Y 122.586,Z 600.869,A -85,B 0,C 180,E1 -25631.622,E2 -25631.622} C_VEL
LIN {X 0,Y 121.262,Z 605.95,A -85,B 0,C 180,E1 -25634.884,E2 -25634.884} C_VEL
LIN {X 0,Y 120.339,Z 610.174,A -85,B 0,C 180,E1 -25638.207,E2 -25638.207} C_VEL
LIN {X 0,Y 119.739,Z 613.654,A -85,B 0,C 180,E1 -25641.564,E2 -25641.564} C_VEL
LIN {X 0,Y 119.424,Z 617.605,A -85,B 0,C 180,E1 -25646.628,E2 -25646.628} C_VEL
LIN {X 0,Y 119.475,Z 619.493,A -85,B 0,C 180,E1 -25650.002,E2 -25650.002} C_VEL
LIN {X 0,Y 119.362,Z 620.842,A -85,B 0,C 180,E1 -25653.377,E2 -25653.377} C_VEL
LIN {X 0,Y 119.54,Z 621.696,A -85,B 0,C 180,E1 -25656.754,E2 -25656.754} C_VEL
LIN {X 0,Y 120.044,Z 621.975,A -85,B 0,C 180,E1 -25660.117,E2 -25660.117} C_VEL
LIN {X 0,Y 120.93,Z 621.784,A -85,B 0,C 180,E1 -25663.444,E2 -25663.444} C_VEL
LIN {X 0,Y 122.256,Z 621.151,A -85,B 0,C 180,E1 -25666.706,E2 -25666.706} C_VEL
LIN {X 0,Y 123.967,Z 620.067,A -85,B 0,C 180,E1 -25669.888,E2 -25669.888} C_VEL
LIN {X 0,Y 127.289,Z 617.384,A -85,B 0,C 180,E1 -25674.464,E2 -25674.464} C_VEL
LIN {X 0,Y 131.521,Z 613.499,A -85,B 0,C 180,E1 -25678.748,E2 -25678.748} C_VEL
LIN {X 0,Y 136.363,Z 608.729,A -85,B 0,C 180,E1 -25682.326,E2 -25682.326} C_VEL
LIN {X 0,Y 136.856,Z 608.575,A -85,B 0,C 180,E1 -25682.632,E2 -25682.632} C_VEL
LIN {X 0,Y 142.447,Z 609.916,A -85,B 0,C 180,E1 -25686.305,E2 -25686.305} C_VEL
LIN {X 0,Y 151.264,Z 610.664,A -85,B 0,C 180,E1 -25690.578,E2 -25690.578} C_VEL
LIN {X 0,Y 155.195,Z 610.503,A -85,B 0,C 180,E1 -25692.789,E2 -25692.789} C_VEL
LIN {X 0,Y 156.675,Z 610.336,A -85,B 0,C 180,E1 -25694.134,E2 -25694.134} C_VEL
LIN {X 0,Y 157.25,Z 610.073,A -85,B 0,C 180,E1 -25695.652,E2 -25695.652} C_VEL
LIN {X 0,Y 157.61,Z 609.632,A -85,B 0,C 180,E1 -25698.021,E2 -25698.021} C_VEL
LIN {X 0,Y 157.485,Z 609.375,A -85,B 0,C 180,E1 -25699.347,E2 -25699.347} C_VEL
LIN {X 0,Y 155.645,Z 609.016,A -85,B 0,C 180,E1 -25700.791,E2 -25700.791} C_VEL
LIN {X 0,Y 150.904,Z 608.423,A -85,B 0,C 180,E1 -25702.74,E2 -25702.74} C_VEL
LIN {X 0,Y 142.143,Z 606.034,A -85,B 0,C 180,E1 -25707.053,E2 -25707.053} C_VEL
LIN {X 0,Y 136.502,Z 603.391,A -85,B 0,C 180,E1 -25710.717,E2 -25710.717} C_VEL
LIN {X 0,Y 131.687,Z 599.968,A -85,B 0,C 180,E1 -25714.726,E2 -25714.726} C_VEL
LIN {X 0,Y 127.743,Z 595.668,A -85,B 0,C 180,E1 -25719.047,E2 -25719.047} C_VEL
LIN {X 0,Y 124.957,Z 590.505,A -85,B 0,C 180,E1 -25723.667,E2 -25723.667} C_VEL
LIN {X 0,Y 123.685,Z 586.246,A -85,B 0,C 180,E1 -25727.176,E2 -25727.176} C_VEL
LIN {X 0,Y 122.989,Z 587.261,A -85,B 0,C 180,E1 -25728.463,E2 -25728.463} C_VEL
LIN {X 0,Y 123.088,Z 587.674,A -85,B 0,C 180,E1 -25730.532,E2 -25730.532} C_VEL
LIN {X 0,Y 123.338,Z 588.321,A -85,B 0,C 180,E1 -25733.259,E2 -25733.259} C_VEL
LIN {X 0,Y 122.76,Z 590.861,A -85,B 0,C 180,E1 -25737.729,E2 -25737.729} C_VEL
LIN {X 0,Y 122.919,Z 593.45,A -85,B 0,C 180,E1 -25742.215,E2 -25742.215} C_VEL
LIN {X 0,Y 124.329,Z 594.11,A -85,B 0,C 180,E1 -25744.856,E2 -25744.856} C_VEL
LIN {X 0,Y 138.406,Z 594.686,A -85,B 0,C 180,E1 -25756.255,E2 -25756.255} C_VEL
LIN {X 0,Y 139.194,Z 594.894,A -85,B 0,C 180,E1 -25756.877,E2 -25756.877} C_VEL
LIN {X 0,Y 136.173,Z 598.877,A -85,B 0,C 180,E1 -25758.837,E2 -25758.837} C_VEL
LIN {X 0,Y 131.378,Z 604.088,A -85,B 0,C 180,E1 -25761.991,E2 -25761.991} C_VEL
LIN {X 0,Y 127.743,Z 607.64,A -85,B 0,C 180,E1 -25764.797,E2 -25764.797} C_VEL
LIN {X 0,Y 123.843,Z 610.991,A -85,B 0,C 180,E1 -25768.401,E2 -25768.401} C_VEL
LIN {X 0,Y 121.033,Z 613.12,A -85,B 0,C 180,E1 -25771.507,E2 -25771.507} C_VEL
LIN {X 0,Y 117.176,Z 615.299,A -85,B 0,C 180,E1 -25776.854,E2 -25776.854} C_VEL
LIN {X 0,Y 114.363,Z 616.187,A -85,B 0,C 180,E1 -25782.531,E2 -25782.531} C_VEL
LIN {X 0,Y 112.545,Z 615.725,A -85,B 0,C 180,E1 -25788.535,E2 -25788.535} C_VEL
LIN {X 0,Y 111.744,Z 613.32,A -85,B 0,C 180,E1 -25795.523,E2 -25795.523} C_VEL
LIN {X 0,Y 112.172,Z 609.948,A -85,B 0,C 180,E1 -25801.301,E2 -25801.301} C_VEL
LIN {X 0,Y 113.345,Z 604.7,A -85,B 0,C 180,E1 -25807.199,E2 -25807.199} C_VEL
LIN {X 0,Y 114.579,Z 599.975,A -85,B 0,C 180,E1 -25811.213,E2 -25811.213} C_VEL
LIN {X 0,Y 116.257,Z 593.906,A -85,B 0,C 180,E1 -25815.294,E2 -25815.294} C_VEL
LIN {X 0,Y 118.278,Z 587.185,A -85,B 0,C 180,E1 -25818.864,E2 -25818.864} C_VEL
LIN {X 0,Y 121.01,Z 577.526,A -85,B 0,C 180,E1 -25822.791,E2 -25822.791} C_VEL
LIN {X 0,Y 121.422,Z 574.769,A -85,B 0,C 180,E1 -25823.751,E2 -25823.751} C_VEL
LIN {X 0,Y 121.259,Z 566.025,A -85,B 0,C 180,E1 -25826.676,E2 -25826.676} C_VEL
LIN {X 0,Y 120.476,Z 554.837,A -85,B 0,C 180,E1 -25829.723,E2 -25829.723} C_VEL
LIN {X 0,Y 119.181,Z 545.132,A -85,B 0,C 180,E1 -25831.898,E2 -25831.898} C_VEL
LIN {X 0,Y 117.461,Z 537.186,A -85,B 0,C 180,E1 -25833.485,E2 -25833.485} C_VEL
LIN {X 0,Y 115.965,Z 533.388,A -85,B 0,C 180,E1 -25834.343,E2 -25834.343} C_VEL
LIN {X 0,Y 115.418,Z 530.922,A -85,B 0,C 180,E1 -25837.873,E2 -25837.873} C_VEL
LIN {X 0,Y 115.287,Z 530.937,A -85,B 0,C 180,E1 -25842.741,E2 -25842.741} C_VEL
LIN {X 0,Y 115.019,Z 530.97,A -85,B 0,C 180,E1 -25847.787,E2 -25847.787} C_VEL
LIN {X 0,Y 114.947,Z 530.974,A -85,B 0,C 180,E1 -25853.491,E2 -25853.491} C_VEL
LIN {X 0,Y 114.869,Z 530.989,A -85,B 0,C 180,E1 -25861.067,E2 -25861.067} C_VEL
LIN {X 0,Y 114.841,Z 530.992,A -85,B 0,C 180,E1 -25867.73,E2 -25867.73} C_VEL
LIN {X 0,Y 114.86,Z 530.979,A -85,B 0,C 180,E1 -25872.756,E2 -25872.756} C_VEL
LIN {X 0,Y 114.868,Z 530.989,A -85,B 0,C 180,E1 -25877.699,E2 -25877.699} C_VEL
LIN {X 0,Y 114.853,Z 530.977,A -85,B 0,C 180,E1 -25882.698,E2 -25882.698} C_VEL
LIN {X 0,Y 114.867,Z 530.989,A -85,B 0,C 180,E1 -25888.931,E2 -25888.931} C_VEL
LIN {X 0,Y 114.944,Z 530.979,A -85,B 0,C 180,E1 -25896.507,E2 -25896.507} C_VEL
LIN {X 0,Y 115.016,Z 530.967,A -85,B 0,C 180,E1 -25902.21,E2 -25902.21} C_VEL
LIN {X 0,Y 115.284,Z 530.935,A -85,B 0,C 180,E1 -25907.257,E2 -25907.257} C_VEL
LIN {X 0,Y 115.396,Z 530.923,A -85,B 0,C 180,E1 -25913.003,E2 -25913.003} C_VEL
LIN {X 0,Y 115.994,Z 530.837,A -85,B 0,C 180,E1 -25920,E2 -25920} C_VEL
LIN {X 0,Y 115.396,Z 530.92,A -85,B 0,C 180,E1 -25926.996,E2 -25926.996} C_VEL
LIN {X 0,Y 115.391,Z 530.923,A -85,B 0,C 180,E1 -25930.528,E2 -25930.528} C_VEL
LIN {X 0,Y 115.146,Z 530.956,A -85,B 0,C 180,E1 -25934.131,E2 -25934.131} C_VEL
LIN {X 0,Y 114.978,Z 530.977,A -85,B 0,C 180,E1 -25941.515,E2 -25941.515} C_VEL
LIN {X 0,Y 114.868,Z 530.991,A -85,B 0,C 180,E1 -25945.358,E2 -25945.358} C_VEL
LIN {X 0,Y 114.866,Z 530.991,A -85,B 0,C 180,E1 -25951.069,E2 -25951.069} C_VEL
LIN {X 0,Y 114.811,Z 530.993,A -85,B 0,C 180,E1 -25957.744,E2 -25957.744} C_VEL
LIN {X 0,Y 114.846,Z 530.994,A -85,B 0,C 180,E1 -25962.751,E2 -25962.751} C_VEL
LIN {X 0,Y 114.949,Z 531.132,A -85,B 0,C 180,E1 -25967.443,E2 -25967.443} C_VEL
LIN {X 0,Y 116.55,Z 536.302,A -85,B 0,C 180,E1 -25971.836,E2 -25971.836} C_VEL
LIN {X 0,Y 119.229,Z 542.56,A -85,B 0,C 180,E1 -25973.166,E2 -25973.166} C_VEL
LIN {X 0,Y 120.432,Z 553.881,A -85,B 0,C 180,E1 -25975.065,E2 -25975.065} C_VEL
LIN {X 0,Y 120.777,Z 564.64,A -85,B 0,C 180,E1 -25977.404,E2 -25977.404} C_VEL
LIN {X 0,Y 120.467,Z 573.284,A -85,B 0,C 180,E1 -25979.693,E2 -25979.693} C_VEL
LIN {X 0,Y 119.846,Z 581.94,A -85,B 0,C 180,E1 -25982.498,E2 -25982.498} C_VEL
LIN {X 0,Y 119.22,Z 587.677,A -85,B 0,C 180,E1 -25984.7,E2 -25984.7} C_VEL
LIN {X 0,Y 117.663,Z 593.369,A -85,B 0,C 180,E1 -25987.157,E2 -25987.157} C_VEL
LIN {X 0,Y 115.821,Z 599.684,A -85,B 0,C 180,E1 -25990.506,E2 -25990.506} C_VEL
LIN {X 0,Y 114.419,Z 604.939,A -85,B 0,C 180,E1 -25993.956,E2 -25993.956} C_VEL
LIN {X 0,Y 113.389,Z 609.312,A -85,B 0,C 180,E1 -25997.473,E2 -25997.473} C_VEL
LIN {X 0,Y 112.533,Z 614.423,A -85,B 0,C 180,E1 -26002.827,E2 -26002.827} C_VEL
LIN {X 0,Y 112.342,Z 617.008,A -85,B 0,C 180,E1 -26006.415,E2 -26006.415} C_VEL
LIN {X 0,Y 112.409,Z 619.018,A -85,B 0,C 180,E1 -26010.002,E2 -26010.002} C_VEL
LIN {X 0,Y 112.29,Z 620.476,A -85,B 0,C 180,E1 -26013.59,E2 -26013.59} C_VEL
LIN {X 0,Y 112.486,Z 621.359,A -85,B 0,C 180,E1 -26017.18,E2 -26017.18} C_VEL
LIN {X 0,Y 113.06,Z 621.724,A -85,B 0,C 180,E1 -26020.75,E2 -26020.75} C_VEL
LIN {X 0,Y 114.029,Z 621.65,A -85,B 0,C 180,E1 -26024.274,E2 -26024.274} C_VEL
LIN {X 0,Y 115.455,Z 621.139,A -85,B 0,C 180,E1 -26027.722,E2 -26027.722} C_VEL
LIN {X 0,Y 117.312,Z 620.138,A -85,B 0,C 180,E1 -26031.068,E2 -26031.068} C_VEL
LIN {X 0,Y 120.865,Z 617.629,A -85,B 0,C 180,E1 -26035.857,E2 -26035.857} C_VEL
LIN {X 0,Y 125.363,Z 613.88,A -85,B 0,C 180,E1 -26040.303,E2 -26040.303} C_VEL
LIN {X 0,Y 130.944,Z 608.792,A -85,B 0,C 180,E1 -26044.304,E2 -26044.304} C_VEL
LIN {X 0,Y 132.485,Z 607.354,A -85,B 0,C 180,E1 -26045.234,E2 -26045.234} C_VEL
LIN {X 0,Y 141.228,Z 609.359,A -85,B 0,C 180,E1 -26050.312,E2 -26050.312} C_VEL
LIN {X 0,Y 145.931,Z 609.788,A -85,B 0,C 180,E1 -26052.397,E2 -26052.397} C_VEL
LIN {X 0,Y 149.701,Z 609.879,A -85,B 0,C 180,E1 -26054.767,E2 -26054.767} C_VEL
LIN {X 0,Y 150.47,Z 609.271,A -85,B 0,C 180,E1 -26058.36,E2 -26058.36} C_VEL
LIN {X 0,Y 150.046,Z 609.123,A -85,B 0,C 180,E1 -26059.024,E2 -26059.024} C_VEL
LIN {X 0,Y 139.62,Z 606.526,A -85,B 0,C 180,E1 -26063.65,E2 -26063.65} C_VEL
LIN {X 0,Y 132.309,Z 603.317,A -85,B 0,C 180,E1 -26067.915,E2 -26067.915} C_VEL
LIN {X 0,Y 127,Z 599.76,A -85,B 0,C 180,E1 -26071.941,E2 -26071.941} C_VEL
LIN {X 0,Y 122.647,Z 595.402,A -85,B 0,C 180,E1 -26076.352,E2 -26076.352} C_VEL
LIN {X 0,Y 119.484,Z 590.726,A -85,B 0,C 180,E1 -26080.731,E2 -26080.731} C_VEL
LIN {X 0,Y 118.194,Z 591.736,A -85,B 0,C 180,E1 -26082.704,E2 -26082.704} C_VEL
LIN {X 0,Y 118.177,Z 591.714,A -85,B 0,C 180,E1 -26086.239,E2 -26086.239} C_VEL
LIN {X 0,Y 117.851,Z 592.503,A -85,B 0,C 180,E1 -26089.694,E2 -26089.694} C_VEL
LIN {X 0,Y 119.881,Z 592.946,A -85,B 0,C 180,E1 -26096.639,E2 -26096.639} C_VEL
LIN {X 0,Y 123.076,Z 594.013,A -85,B 0,C 180,E1 -26103.274,E2 -26103.274} C_VEL
LIN {X 0,Y 124.329,Z 594.11,A -85,B 0,C 180,E1 -26104.856,E2 -26104.856} C_VEL
LIN {X 0,Y 125.314,Z 594.629,A -85,B 0,C 180,E1 -26106.614,E2 -26106.614} C_VEL
LIN {X 0,Y 126.787,Z 598.396,A -85,B 0,C 180,E1 -26112.463,E2 -26112.463} C_VEL
LIN {X 0,Y 128.326,Z 598.842,A -85,B 0,C 180,E1 -26114.094,E2 -26114.094} C_VEL
LIN {X 0,Y 131.535,Z 598.952,A -85,B 0,C 180,E1 -26116.291,E2 -26116.291} C_VEL
LIN {X 0,Y 126.718,Z 604.059,A -85,B 0,C 180,E1 -26119.459,E2 -26119.459} C_VEL
LIN {X 0,Y 122.038,Z 608.231,A -85,B 0,C 180,E1 -26122.862,E2 -26122.862} C_VEL
LIN {X 0,Y 117.882,Z 611.474,A -85,B 0,C 180,E1 -26126.579,E2 -26126.579} C_VEL
LIN {X 0,Y 114.219,Z 613.85,A -85,B 0,C 180,E1 -26130.519,E2 -26130.519} C_VEL
LIN {X 0,Y 111.126,Z 615.436,A -85,B 0,C 180,E1 -26134.694,E2 -26134.694} C_VEL
LIN {X 0,Y 107.888,Z 616.371,A -85,B 0,C 180,E1 -26140.649,E2 -26140.649} C_VEL
LIN {X 0,Y 105.767,Z 615.989,A -85,B 0,C 180,E1 -26146.964,E2 -26146.964} C_VEL
LIN {X 0,Y 104.736,Z 613.992,A -85,B 0,C 180,E1 -26153.633,E2 -26153.633} C_VEL
LIN {X 0,Y 104.685,Z 612.198,A -85,B 0,C 180,E1 -26157.513,E2 -26157.513} C_VEL
LIN {X 0,Y 105.18,Z 609.297,A -85,B 0,C 180,E1 -26162.111,E2 -26162.111} C_VEL
LIN {X 0,Y 106.323,Z 604.421,A -85,B 0,C 180,E1 -26167.73,E2 -26167.73} C_VEL
LIN {X 0,Y 108.021,Z 598.36,A -85,B 0,C 180,E1 -26172.974,E2 -26172.974} C_VEL
LIN {X 0,Y 110.407,Z 590.428,A -85,B 0,C 180,E1 -26178.059,E2 -26178.059} C_VEL
LIN {X 0,Y 112.564,Z 583.369,A -85,B 0,C 180,E1 -26181.517,E2 -26181.517} C_VEL
LIN {X 0,Y 114.568,Z 576.36,A -85,B 0,C 180,E1 -26184.277,E2 -26184.277} C_VEL
LIN {X 0,Y 114.59,Z 568.909,A -85,B 0,C 180,E1 -26187.016,E2 -26187.016} C_VEL
LIN {X 0,Y 114.239,Z 560.53,A -85,B 0,C 180,E1 -26189.652,E2 -26189.652} C_VEL
LIN {X 0,Y 113.361,Z 551.156,A -85,B 0,C 180,E1 -26192.16,E2 -26192.16} C_VEL
LIN {X 0,Y 111.604,Z 540.545,A -85,B 0,C 180,E1 -26194.58,E2 -26194.58} C_VEL
LIN {X 0,Y 108.692,Z 533.503,A -85,B 0,C 180,E1 -26196.379,E2 -26196.379} C_VEL
LIN {X 0,Y 108.401,Z 531.796,A -85,B 0,C 180,E1 -26198.856,E2 -26198.856} C_VEL
LIN {X 0,Y 108.04,Z 531.839,A -85,B 0,C 180,E1 -26205.08,E2 -26205.08} C_VEL
LIN {X 0,Y 107.911,Z 531.85,A -85,B 0,C 180,E1 -26213,E2 -26213} C_VEL
LIN {X 0,Y 107.807,Z 531.868,A -85,B 0,C 180,E1 -26221.432,E2 -26221.432} C_VEL
LIN {X 0,Y 107.749,Z 531.876,A -85,B 0,C 180,E1 -26228.49,E2 -26228.49} C_VEL
LIN {X 0,Y 107.766,Z 531.871,A -85,B 0,C 180,E1 -26235.835,E2 -26235.835} C_VEL
LIN {X 0,Y 107.753,Z 531.865,A -85,B 0,C 180,E1 -26241.503,E2 -26241.503} C_VEL
LIN {X 0,Y 107.808,Z 531.868,A -85,B 0,C 180,E1 -26248.566,E2 -26248.566} C_VEL
LIN {X 0,Y 107.908,Z 531.855,A -85,B 0,C 180,E1 -26256.997,E2 -26256.997} C_VEL
LIN {X 0,Y 108.037,Z 531.839,A -85,B 0,C 180,E1 -26264.917,E2 -26264.917} C_VEL
LIN {X 0,Y 108.291,Z 531.801,A -85,B 0,C 180,E1 -26268.773,E2 -26268.773} C_VEL
LIN {X 0,Y 108.461,Z 531.78,A -85,B 0,C 180,E1 -26276.284,E2 -26276.284} C_VEL
LIN {X 0,Y 108.945,Z 531.714,A -85,B 0,C 180,E1 -26280,E2 -26280} C_VEL
LIN {X 0,Y 108.338,Z 531.8,A -85,B 0,C 180,E1 -26287.454,E2 -26287.454} C_VEL
LIN {X 0,Y 108.2,Z 531.819,A -85,B 0,C 180,E1 -26293.026,E2 -26293.026} C_VEL
LIN {X 0,Y 107.906,Z 531.859,A -85,B 0,C 180,E1 -26299.005,E2 -26299.005} C_VEL
LIN {X 0,Y 107.855,Z 531.865,A -85,B 0,C 180,E1 -26304.185,E2 -26304.185} C_VEL
LIN {X 0,Y 107.792,Z 531.872,A -85,B 0,C 180,E1 -26312.053,E2 -26312.053} C_VEL
LIN {X 0,Y 107.723,Z 531.877,A -85,B 0,C 180,E1 -26318.476,E2 -26318.476} C_VEL
LIN {X 0,Y 107.801,Z 531.937,A -85,B 0,C 180,E1 -26325.818,E2 -26325.818} C_VEL
LIN {X 0,Y 109.056,Z 536.134,A -85,B 0,C 180,E1 -26329.794,E2 -26329.794} C_VEL
LIN {X 0,Y 113.014,Z 544.994,A -85,B 0,C 180,E1 -26331.909,E2 -26331.909} C_VEL
LIN {X 0,Y 113.926,Z 555.958,A -85,B 0,C 180,E1 -26334.015,E2 -26334.015} C_VEL
LIN {X 0,Y 114.161,Z 564.096,A -85,B 0,C 180,E1 -26335.924,E2 -26335.924} C_VEL
LIN {X 0,Y 113.727,Z 573.351,A -85,B 0,C 180,E1 -26338.523,E2 -26338.523} C_VEL
LIN {X 0,Y 113.071,Z 581.205,A -85,B 0,C 180,E1 -26341.205,E2 -26341.205} C_VEL
LIN {X 0,Y 112.248,Z 588.075,A -85,B 0,C 180,E1 -26344.008,E2 -26344.008} C_VEL
LIN {X 0,Y 110.064,Z 595.322,A -85,B 0,C 180,E1 -26347.475,E2 -26347.475} C_VEL
LIN {X 0,Y 107.969,Z 602.687,A -85,B 0,C 180,E1 -26351.992,E2 -26351.992} C_VEL
LIN {X 0,Y 106.466,Z 608.45,A -85,B 0,C 180,E1 -26356.644,E2 -26356.644} C_VEL
LIN {X 0,Y 105.707,Z 612.182,A -85,B 0,C 180,E1 -26360.434,E2 -26360.434} C_VEL
LIN {X 0,Y 105.255,Z 616.404,A -85,B 0,C 180,E1 -26366.173,E2 -26366.173} C_VEL
LIN {X 0,Y 105.333,Z 618.533,A -85,B 0,C 180,E1 -26370.002,E2 -26370.002} C_VEL
LIN {X 0,Y 105.223,Z 620.042,A -85,B 0,C 180,E1 -26373.832,E2 -26373.832} C_VEL
LIN {X 0,Y 105.457,Z 620.983,A -85,B 0,C 180,E1 -26377.662,E2 -26377.662} C_VEL
LIN {X 0,Y 106.103,Z 621.47,A -85,B 0,C 180,E1 -26381.464,E2 -26381.464} C_VEL
LIN {X 0,Y 107.163,Z 621.518,A -85,B 0,C 180,E1 -26385.21,E2 -26385.21} C_VEL
LIN {X 0,Y 108.697,Z 621.112,A -85,B 0,C 180,E1 -26388.864,E2 -26388.864} C_VEL
LIN {X 0,Y 110.718,Z 620.14,A -85,B 0,C 180,E1 -26392.389,E2 -26392.389} C_VEL
LIN {X 0,Y 113.116,Z 618.683,A -85,B 0,C 180,E1 -26395.782,E2 -26395.782} C_VEL
LIN {X 0,Y 117.647,Z 615.61,A -85,B 0,C 180,E1 -26400.517,E2 -26400.517} C_VEL
LIN {X 0,Y 123.154,Z 611.246,A -85,B 0,C 180,E1 -26404.799,E2 -26404.799} C_VEL
LIN {X 0,Y 128.821,Z 606.14,A -85,B 0,C 180,E1 -26408.236,E2 -26408.236} C_VEL
LIN {X 0,Y 136.005,Z 607.94,A -85,B 0,C 180,E1 -26412.206,E2 -26412.206} C_VEL
LIN {X 0,Y 140.719,Z 608.725,A -85,B 0,C 180,E1 -26414.366,E2 -26414.366} C_VEL
LIN {X 0,Y 143.072,Z 608.712,A -85,B 0,C 180,E1 -26416.551,E2 -26416.551} C_VEL
LIN {X 0,Y 143.215,Z 608.573,A -85,B 0,C 180,E1 -26417.402,E2 -26417.402} C_VEL
LIN {X 0,Y 139.867,Z 607.682,A -85,B 0,C 180,E1 -26419.216,E2 -26419.216} C_VEL
LIN {X 0,Y 130.55,Z 604.222,A -85,B 0,C 180,E1 -26423.689,E2 -26423.689} C_VEL
LIN {X 0,Y 124.508,Z 600.802,A -85,B 0,C 180,E1 -26427.572,E2 -26427.572} C_VEL
LIN {X 0,Y 119.345,Z 596.631,A -85,B 0,C 180,E1 -26431.894,E2 -26431.894} C_VEL
LIN {X 0,Y 117.389,Z 594.602,A -85,B 0,C 180,E1 -26433.906,E2 -26433.906} C_VEL
LIN {X 0,Y 116.2,Z 595.274,A -85,B 0,C 180,E1 -26434.953,E2 -26434.953} C_VEL
LIN {X 0,Y 115.357,Z 595.634,A -85,B 0,C 180,E1 -26436.048,E2 -26436.048} C_VEL
LIN {X 0,Y 113.069,Z 596.355,A -85,B 0,C 180,E1 -26441.894,E2 -26441.894} C_VEL
LIN {X 0,Y 112.833,Z 596.403,A -85,B 0,C 180,E1 -26445.573,E2 -26445.573} C_VEL
LIN {X 0,Y 112.456,Z 596.99,A -85,B 0,C 180,E1 -26449.194,E2 -26449.194} C_VEL
LIN {X 0,Y 114.225,Z 597.403,A -85,B 0,C 180,E1 -26456.473,E2 -26456.473} C_VEL
LIN {X 0,Y 117.352,Z 598.325,A -85,B 0,C 180,E1 -26463.434,E2 -26463.434} C_VEL
LIN {X 0,Y 128.326,Z 598.842,A -85,B 0,C 180,E1 -26474.094,E2 -26474.094} C_VEL
LIN {X 0,Y 128.742,Z 599.293,A -85,B 0,C 180,E1 -26474.908,E2 -26474.908} C_VEL
LIN {X 0,Y 128.092,Z 600.503,A -85,B 0,C 180,E1 -26475.904,E2 -26475.904} C_VEL
LIN {X 0,Y 125.972,Z 602.589,A -85,B 0,C 180,E1 -26477.076,E2 -26477.076} C_VEL
LIN {X 0,Y 118.198,Z 607.735,A -85,B 0,C 180,E1 -26479.769,E2 -26479.769} C_VEL
LIN {X 0,Y 116.343,Z 608.948,A -85,B 0,C 180,E1 -26480.86,E2 -26480.86} C_VEL
LIN {X 0,Y 112.042,Z 611.982,A -85,B 0,C 180,E1 -26484.559,E2 -26484.559} C_VEL
LIN {X 0,Y 110.018,Z 613.302,A -85,B 0,C 180,E1 -26486.574,E2 -26486.574} C_VEL
LIN {X 0,Y 105.268,Z 615.581,A -85,B 0,C 180,E1 -26492.283,E2 -26492.283} C_VEL
LIN {X 0,Y 103.313,Z 616.289,A -85,B 0,C 180,E1 -26495.279,E2 -26495.279} C_VEL
LIN {X 0,Y 100.887,Z 616.651,A -85,B 0,C 180,E1 -26499.976,E2 -26499.976} C_VEL
LIN {X 0,Y 99.048,Z 616.238,A -85,B 0,C 180,E1 -26505.199,E2 -26505.199} C_VEL
LIN {X 0,Y 97.755,Z 614.341,A -85,B 0,C 180,E1 -26512.264,E2 -26512.264} C_VEL
LIN {X 0,Y 97.577,Z 612.119,A -85,B 0,C 180,E1 -26517.304,E2 -26517.304} C_VEL
LIN {X 0,Y 98.098,Z 609.126,A -85,B 0,C 180,E1 -26522.244,E2 -26522.244} C_VEL
LIN {X 0,Y 99.076,Z 605.115,A -85,B 0,C 180,E1 -26527.244,E2 -26527.244} C_VEL
LIN {X 0,Y 100.278,Z 600.656,A -85,B 0,C 180,E1 -26531.614,E2 -26531.614} C_VEL
LIN {X 0,Y 101.72,Z 596.022,A -85,B 0,C 180,E1 -26535.304,E2 -26535.304} C_VEL
LIN {X 0,Y 103.7,Z 589.856,A -85,B 0,C 180,E1 -26539.257,E2 -26539.257} C_VEL
LIN {X 0,Y 105.645,Z 583.885,A -85,B 0,C 180,E1 -26542.352,E2 -26542.352} C_VEL
LIN {X 0,Y 107.763,Z 576.784,A -85,B 0,C 180,E1 -26545.337,E2 -26545.337} C_VEL
LIN {X 0,Y 107.851,Z 569.695,A -85,B 0,C 180,E1 -26548.131,E2 -26548.131} C_VEL
LIN {X 0,Y 107.6,Z 561.396,A -85,B 0,C 180,E1 -26550.933,E2 -26550.933} C_VEL
LIN {X 0,Y 106.864,Z 552.357,A -85,B 0,C 180,E1 -26553.545,E2 -26553.545} C_VEL
LIN {X 0,Y 105.502,Z 543.426,A -85,B 0,C 180,E1 -26555.805,E2 -26555.805} C_VEL
LIN {X 0,Y 101.528,Z 533.594,A -85,B 0,C 180,E1 -26558.707,E2 -26558.707} C_VEL
LIN {X 0,Y 101.283,Z 532.683,A -85,B 0,C 180,E1 -26560.493,E2 -26560.493} C_VEL
LIN {X 0,Y 100.93,Z 532.723,A -85,B 0,C 180,E1 -26566.17,E2 -26566.17} C_VEL
LIN {X 0,Y 100.819,Z 532.737,A -85,B 0,C 180,E1 -26570.396,E2 -26570.396} C_VEL
LIN {X 0,Y 100.774,Z 532.743,A -85,B 0,C 180,E1 -26574.956,E2 -26574.956} C_VEL
LIN {X 0,Y 100.703,Z 532.751,A -85,B 0,C 180,E1 -26583.126,E2 -26583.126} C_VEL
LIN {X 0,Y 100.696,Z 532.752,A -85,B 0,C 180,E1 -26589.848,E2 -26589.848} C_VEL
LIN {X 0,Y 100.732,Z 532.747,A -85,B 0,C 180,E1 -26595.757,E2 -26595.757} C_VEL
LIN {X 0,Y 100.694,Z 532.747,A -85,B 0,C 180,E1 -26601.085,E2 -26601.085} C_VEL
LIN {X 0,Y 100.705,Z 532.751,A -85,B 0,C 180,E1 -26606.868,E2 -26606.868} C_VEL
LIN {X 0,Y 100.784,Z 532.741,A -85,B 0,C 180,E1 -26615.266,E2 -26615.266} C_VEL
LIN {X 0,Y 100.816,Z 532.735,A -85,B 0,C 180,E1 -26619.601,E2 -26619.601} C_VEL
LIN {X 0,Y 101.189,Z 532.687,A -85,B 0,C 180,E1 -26627.973,E2 -26627.973} C_VEL
LIN {X 0,Y 101.272,Z 532.683,A -85,B 0,C 180,E1 -26632.022,E2 -26632.022} C_VEL
LIN {X 0,Y 101.869,Z 532.595,A -85,B 0,C 180,E1 -26640,E2 -26640} C_VEL
LIN {X 0,Y 101.277,Z 532.681,A -85,B 0,C 180,E1 -26647.977,E2 -26647.977} C_VEL
LIN {X 0,Y 101.126,Z 532.701,A -85,B 0,C 180,E1 -26653.363,E2 -26653.363} C_VEL
LIN {X 0,Y 100.816,Z 532.741,A -85,B 0,C 180,E1 -26660.399,E2 -26660.399} C_VEL
LIN {X 0,Y 100.771,Z 532.747,A -85,B 0,C 180,E1 -26664.959,E2 -26664.959} C_VEL
LIN {X 0,Y 100.698,Z 532.756,A -85,B 0,C 180,E1 -26673.126,E2 -26673.126} C_VEL
LIN {X 0,Y 100.675,Z 532.759,A -85,B 0,C 180,E1 -26679.838,E2 -26679.838} C_VEL
LIN {X 0,Y 100.763,Z 532.946,A -85,B 0,C 180,E1 -26684.225,E2 -26684.225} C_VEL
LIN {X 0,Y 101.654,Z 536.143,A -85,B 0,C 180,E1 -26687.456,E2 -26687.456} C_VEL
LIN {X 0,Y 106.75,Z 547.488,A -85,B 0,C 180,E1 -26690.612,E2 -26690.612} C_VEL
LIN {X 0,Y 107.4,Z 557.166,A -85,B 0,C 180,E1 -26692.707,E2 -26692.707} C_VEL
LIN {X 0,Y 107.542,Z 564.402,A -85,B 0,C 180,E1 -26694.553,E2 -26694.553} C_VEL
LIN {X 0,Y 107.046,Z 573.277,A -85,B 0,C 180,E1 -26697.207,E2 -26697.207} C_VEL
LIN {X 0,Y 106.335,Z 580.895,A -85,B 0,C 180,E1 -26699.962,E2 -26699.962} C_VEL
LIN {X 0,Y 105.537,Z 587.394,A -85,B 0,C 180,E1 -26702.755,E2 -26702.755} C_VEL
LIN {X 0,Y 103.541,Z 593.889,A -85,B 0,C 180,E1 -26705.969,E2 -26705.969} C_VEL
LIN {X 0,Y 101.646,Z 600.056,A -85,B 0,C 180,E1 -26709.777,E2 -26709.777} C_VEL
LIN {X 0,Y 100.106,Z 605.162,A -85,B 0,C 180,E1 -26713.693,E2 -26713.693} C_VEL
LIN {X 0,Y 99.094,Z 609.417,A -85,B 0,C 180,E1 -26717.718,E2 -26717.718} C_VEL
LIN {X 0,Y 98.278,Z 614.408,A -85,B 0,C 180,E1 -26723.844,E2 -26723.844} C_VEL
LIN {X 0,Y 98.244,Z 617.989,A -85,B 0,C 180,E1 -26730.002,E2 -26730.002} C_VEL
LIN {X 0,Y 98.156,Z 619.544,A -85,B 0,C 180,E1 -26734.108,E2 -26734.108} C_VEL
LIN {X 0,Y 98.43,Z 620.606,A -85,B 0,C 180,E1 -26738.212,E2 -26738.212} C_VEL
LIN {X 0,Y 99.146,Z 621.215,A -85,B 0,C 180,E1 -26742.28,E2 -26742.28} C_VEL
LIN {X 0,Y 100.336,Z 621.386,A -85,B 0,C 180,E1 -26746.273,E2 -26746.273} C_VEL
LIN {X 0,Y 101.996,Z 621.018,A -85,B 0,C 180,E1 -26750.155,E2 -26750.155} C_VEL
LIN {X 0,Y 104.173,Z 620.144,A -85,B 0,C 180,E1 -26753.88,E2 -26753.88} C_VEL
LIN {X 0,Y 106.761,Z 618.825,A -85,B 0,C 180,E1 -26757.441,E2 -26757.441} C_VEL
LIN {X 0,Y 111.592,Z 615.893,A -85,B 0,C 180,E1 -26762.368,E2 -26762.368} C_VEL
LIN {X 0,Y 115.315,Z 613.236,A -85,B 0,C 180,E1 -26765.381,E2 -26765.381} C_VEL
LIN {X 0,Y 121.714,Z 608.099,A -85,B 0,C 180,E1 -26769.434,E2 -26769.434} C_VEL
LIN {X 0,Y 125.4,Z 604.837,A -85,B 0,C 180,E1 -26771.323,E2 -26771.323} C_VEL
LIN {X 0,Y 130.96,Z 606.407,A -85,B 0,C 180,E1 -26774.241,E2 -26774.241} C_VEL
LIN {X 0,Y 135.477,Z 607.195,A -85,B 0,C 180,E1 -26776.576,E2 -26776.576} C_VEL
LIN {X 0,Y 134.591,Z 606.86,A -85,B 0,C 180,E1 -26777.248,E2 -26777.248} C_VEL
LIN {X 0,Y 124.979,Z 602.968,A -85,B 0,C 180,E1 -26781.789,E2 -26781.789} C_VEL
LIN {X 0,Y 117.169,Z 598.097,A -85,B 0,C 180,E1 -26786.944,E2 -26786.944} C_VEL
LIN {X 0,Y 113.455,Z 599.186,A -85,B 0,C 180,E1 -26790.294,E2 -26790.294} C_VEL
LIN {X 0,Y 107.686,Z 600.638,A -85,B 0,C 180,E1 -26800.955,E2 -26800.955} C_VEL
LIN {X 0,Y 107.235,Z 600.724,A -85,B 0,C 180,E1 -26804.803,E2 -26804.803} C_VEL
LIN {X 0,Y 106.921,Z 601.252,A -85,B 0,C 180,E1 -26810.4,E2 -26810.4} C_VEL
LIN {X 0,Y 109.591,Z 601.854,A -85,B 0,C 180,E1 -26820,E2 -26820} C_VEL
LIN {X 0,Y 113.863,Z 602.443,A -85,B 0,C 180,E1 -26827.091,E2 -26827.091} C_VEL
LIN {X 0,Y 123.502,Z 602.727,A -85,B 0,C 180,E1 -26835.683,E2 -26835.683} C_VEL
LIN {X 0,Y 122.403,Z 603.957,A -85,B 0,C 180,E1 -26836.684,E2 -26836.684} C_VEL
LIN {X 0,Y 117.102,Z 608.382,A -85,B 0,C 180,E1 -26840.283,E2 -26840.283} C_VEL
LIN {X 0,Y 116.343,Z 608.948,A -85,B 0,C 180,E1 -26840.86,E2 -26840.86} C_VEL
LIN {X 0,Y 112.923,Z 611.128,A -85,B 0,C 180,E1 -26843.031,E2 -26843.031} C_VEL
LIN {X 0,Y 106.097,Z 613.983,A -85,B 0,C 180,E1 -26846.492,E2 -26846.492} C_VEL
LIN {X 0,Y 99.616,Z 615.903,A -85,B 0,C 180,E1 -26850.526,E2 -26850.526} C_VEL
LIN {X 0,Y 96.867,Z 616.418,A -85,B 0,C 180,E1 -26853.546,E2 -26853.546} C_VEL
LIN {X 0,Y 95.401,Z 616.747,A -85,B 0,C 180,E1 -26856.111,E2 -26856.111} C_VEL
LIN {X 0,Y 92.427,Z 616.47,A -85,B 0,C 180,E1 -26863.185,E2 -26863.185} C_VEL
LIN {X 0,Y 90.698,Z 614.312,A -85,B 0,C 180,E1 -26871.688,E2 -26871.688} C_VEL
LIN {X 0,Y 90.471,Z 612.039,A -85,B 0,C 180,E1 -26877.056,E2 -26877.056} C_VEL
LIN {X 0,Y 91.008,Z 608.956,A -85,B 0,C 180,E1 -26882.394,E2 -26882.394} C_VEL
LIN {X 0,Y 91.978,Z 605.06,A -85,B 0,C 180,E1 -26887.537,E2 -26887.537} C_VEL
LIN {X 0,Y 93.354,Z 600.282,A -85,B 0,C 180,E1 -26892.472,E2 -26892.472} C_VEL
LIN {X 0,Y 95.211,Z 594.472,A -85,B 0,C 180,E1 -26897.204,E2 -26897.204} C_VEL
LIN {X 0,Y 98.05,Z 586.339,A -85,B 0,C 180,E1 -26902.31,E2 -26902.31} C_VEL
LIN {X 0,Y 100.934,Z 577.21,A -85,B 0,C 180,E1 -26906.505,E2 -26906.505} C_VEL
LIN {X 0,Y 101.134,Z 570.126,A -85,B 0,C 180,E1 -26909.5,E2 -26909.5} C_VEL
LIN {X 0,Y 101.002,Z 562.01,A -85,B 0,C 180,E1 -26912.452,E2 -26912.452} C_VEL
LIN {X 0,Y 100.368,Z 552.976,A -85,B 0,C 180,E1 -26915.281,E2 -26915.281} C_VEL
LIN {X 0,Y 99.376,Z 546.171,A -85,B 0,C 180,E1 -26917.212,E2 -26917.212} C_VEL
LIN {X 0,Y 95.702,Z 537.169,A -85,B 0,C 180,E1 -26920.163,E2 -26920.163} C_VEL
LIN {X 0,Y 94.265,Z 533.803,A -85,B 0,C 180,E1 -26921.284,E2 -26921.284} C_VEL
LIN {X 0,Y 94.099,Z 533.576,A -85,B 0,C 180,E1 -26922.945,E2 -26922.945} C_VEL
LIN {X 0,Y 93.694,Z 533.623,A -85,B 0,C 180,E1 -26932.025,E2 -26932.025} C_VEL
LIN {X 0,Y 93.623,Z 533.634,A -85,B 0,C 180,E1 -26936.767,E2 -26936.767} C_VEL
LIN {X 0,Y 93.609,Z 533.63,A -85,B 0,C 180,E1 -26944.323,E2 -26944.323} C_VEL
LIN {X 0,Y 93.629,Z 533.623,A -85,B 0,C 180,E1 -26952.494,E2 -26952.494} C_VEL
LIN {X 0,Y 93.627,Z 533.634,A -85,B 0,C 180,E1 -26958.642,E2 -26958.642} C_VEL
LIN {X 0,Y 93.612,Z 533.63,A -85,B 0,C 180,E1 -26965.669,E2 -26965.669} C_VEL
LIN {X 0,Y 93.667,Z 533.625,A -85,B 0,C 180,E1 -26974.203,E2 -26974.203} C_VEL
LIN {X 0,Y 93.692,Z 533.626,A -85,B 0,C 180,E1 -26977.972,E2 -26977.972} C_VEL
LIN {X 0,Y 94.092,Z 533.575,A -85,B 0,C 180,E1 -26987.051,E2 -26987.051} C_VEL
LIN {X 0,Y 94.204,Z 533.562,A -85,B 0,C 180,E1 -26991.419,E2 -26991.419} C_VEL
LIN {X 0,Y 94.795,Z 533.476,A -85,B 0,C 180,E1 -27000,E2 -27000} C_VEL
LIN {X 0,Y 94.209,Z 533.562,A -85,B 0,C 180,E1 -27008.58,E2 -27008.58} C_VEL
LIN {X 0,Y 94.044,Z 533.584,A -85,B 0,C 180,E1 -27013.721,E2 -27013.721} C_VEL
LIN {X 0,Y 93.692,Z 533.63,A -85,B 0,C 180,E1 -27022.028,E2 -27022.028} C_VEL
LIN {X 0,Y 93.62,Z 533.639,A -85,B 0,C 180,E1 -27026.77,E2 -27026.77} C_VEL
LIN {X 0,Y 93.599,Z 533.638,A -85,B 0,C 180,E1 -27034.32,E2 -27034.32} C_VEL
LIN {X 0,Y 93.655,Z 533.697,A -85,B 0,C 180,E1 -27042.105,E2 -27042.105} C_VEL
LIN {X 0,Y 94.236,Z 535.881,A -85,B 0,C 180,E1 -27044.735,E2 -27044.735} C_VEL
LIN {X 0,Y 99.743,Z 548.017,A -85,B 0,C 180,E1 -27048.571,E2 -27048.571} C_VEL
LIN {X 0,Y 100.561,Z 550.187,A -85,B 0,C 180,E1 -27049.254,E2 -27049.254} C_VEL
LIN {X 0,Y 100.973,Z 559.173,A -85,B 0,C 180,E1 -27051.445,E2 -27051.445} C_VEL
LIN {X 0,Y 100.791,Z 569.185,A -85,B 0,C 180,E1 -27054.355,E2 -27054.355} C_VEL
LIN {X 0,Y 99.785,Z 579.374,A -85,B 0,C 180,E1 -27058.057,E2 -27058.057} C_VEL
LIN {X 0,Y 98.634,Z 587.667,A -85,B 0,C 180,E1 -27061.835,E2 -27061.835} C_VEL
LIN {X 0,Y 96.505,Z 594.075,A -85,B 0,C 180,E1 -27065.247,E2 -27065.247} C_VEL
LIN {X 0,Y 94.55,Z 600.181,A -85,B 0,C 180,E1 -27069.327,E2 -27069.327} C_VEL
LIN {X 0,Y 92.975,Z 605.232,A -85,B 0,C 180,E1 -27073.535,E2 -27073.535} C_VEL
LIN {X 0,Y 92.168,Z 608.497,A -85,B 0,C 180,E1 -27076.778,E2 -27076.778} C_VEL
LIN {X 0,Y 91.431,Z 612.151,A -85,B 0,C 180,E1 -27081.159,E2 -27081.159} C_VEL
LIN {X 0,Y 91.118,Z 615.101,A -85,B 0,C 180,E1 -27085.579,E2 -27085.579} C_VEL
LIN {X 0,Y 91.163,Z 617.369,A -85,B 0,C 180,E1 -27090.002,E2 -27090.002} C_VEL
LIN {X 0,Y 91.084,Z 619.034,A -85,B 0,C 180,E1 -27094.428,E2 -27094.428} C_VEL
LIN {X 0,Y 91.402,Z 620.219,A -85,B 0,C 180,E1 -27098.848,E2 -27098.848} C_VEL
LIN {X 0,Y 92.225,Z 620.956,A -85,B 0,C 180,E1 -27103.218,E2 -27103.218} C_VEL
LIN {X 0,Y 93.525,Z 621.196,A -85,B 0,C 180,E1 -27107.495,E2 -27107.495} C_VEL
LIN {X 0,Y 95.359,Z 620.891,A -85,B 0,C 180,E1 -27111.626,E2 -27111.626} C_VEL
LIN {X 0,Y 97.708,Z 620.151,A -85,B 0,C 180,E1 -27115.57,E2 -27115.57} C_VEL
LIN {X 0,Y 100.508,Z 618.967,A -85,B 0,C 180,E1 -27119.308,E2 -27119.308} C_VEL
LIN {X 0,Y 105.671,Z 616.188,A -85,B 0,C 180,E1 -27124.427,E2 -27124.427} C_VEL
LIN {X 0,Y 109.627,Z 613.698,A -85,B 0,C 180,E1 -27127.522,E2 -27127.522} C_VEL
LIN {X 0,Y 116.346,Z 608.751,A -85,B 0,C 180,E1 -27131.644,E2 -27131.644} C_VEL
LIN {X 0,Y 122.544,Z 603.474,A -85,B 0,C 180,E1 -27134.634,E2 -27134.634} C_VEL
LIN {X 0,Y 126.14,Z 604.499,A -85,B 0,C 180,E1 -27136.413,E2 -27136.413} C_VEL
LIN {X 0,Y 119.307,Z 601.324,A -85,B 0,C 180,E1 -27139.888,E2 -27139.888} C_VEL
LIN {X 0,Y 115.208,Z 602.218,A -85,B 0,C 180,E1 -27142.409,E2 -27142.409} C_VEL
LIN {X 0,Y 111.969,Z 602.461,A -85,B 0,C 180,E1 -27145.604,E2 -27145.604} C_VEL
LIN {X 0,Y 108.4,Z 603.27,A -85,B 0,C 180,E1 -27148.757,E2 -27148.757} C_VEL
LIN {X 0,Y 102.031,Z 604.467,A -85,B 0,C 180,E1 -27159.855,E2 -27159.855} C_VEL
LIN {X 0,Y 100.928,Z 604.864,A -85,B 0,C 180,E1 -27167.137,E2 -27167.137} C_VEL
LIN {X 0,Y 107.547,Z 605.959,A -85,B 0,C 180,E1 -27187.51,E2 -27187.51} C_VEL
LIN {X 0,Y 115.294,Z 606.085,A -85,B 0,C 180,E1 -27195.012,E2 -27195.012} C_VEL
LIN {X 0,Y 114.647,Z 606.965,A -85,B 0,C 180,E1 -27196.008,E2 -27196.008} C_VEL
LIN {X 0,Y 108.662,Z 611.16,A -85,B 0,C 180,E1 -27200.327,E2 -27200.327} C_VEL
LIN {X 0,Y 104.889,Z 613.383,A -85,B 0,C 180,E1 -27203.705,E2 -27203.705} C_VEL
LIN {X 0,Y 99.574,Z 615.739,A -85,B 0,C 180,E1 -27209.609,E2 -27209.609} C_VEL
LIN {X 0,Y 96.867,Z 616.418,A -85,B 0,C 180,E1 -27213.546,E2 -27213.546} C_VEL
LIN {X 0,Y 94.367,Z 616.841,A -85,B 0,C 180,E1 -27216.745,E2 -27216.745} C_VEL
LIN {X 0,Y 91.293,Z 616.83,A -85,B 0,C 180,E1 -27219.884,E2 -27219.884} C_VEL
LIN {X 0,Y 85.464,Z 615.635,A -85,B 0,C 180,E1 -27226.598,E2 -27226.598} C_VEL
LIN {X 0,Y 83.794,Z 614.487,A -85,B 0,C 180,E1 -27230.376,E2 -27230.376} C_VEL
LIN {X 0,Y 83.574,Z 614.02,A -85,B 0,C 180,E1 -27231.689,E2 -27231.689} C_VEL
LIN {X 0,Y 83.4,Z 611.615,A -85,B 0,C 180,E1 -27237.426,E2 -27237.426} C_VEL
LIN {X 0,Y 83.907,Z 608.748,A -85,B 0,C 180,E1 -27242.567,E2 -27242.567} C_VEL
LIN {X 0,Y 85.056,Z 604.457,A -85,B 0,C 180,E1 -27248.514,E2 -27248.514} C_VEL
LIN {X 0,Y 86.843,Z 598.787,A -85,B 0,C 180,E1 -27254.539,E2 -27254.539} C_VEL
LIN {X 0,Y 89.04,Z 592.357,A -85,B 0,C 180,E1 -27259.768,E2 -27259.768} C_VEL
LIN {X 0,Y 92.038,Z 584.13,A -85,B 0,C 180,E1 -27264.735,E2 -27264.735} C_VEL
LIN {X 0,Y 94.163,Z 577.594,A -85,B 0,C 180,E1 -27267.859,E2 -27267.859} C_VEL
LIN {X 0,Y 94.463,Z 570.545,A -85,B 0,C 180,E1 -27271.064,E2 -27271.064} C_VEL
LIN {X 0,Y 94.457,Z 562.315,A -85,B 0,C 180,E1 -27274.265,E2 -27274.265} C_VEL
LIN {X 0,Y 93.965,Z 553.52,A -85,B 0,C 180,E1 -27277.218,E2 -27277.218} C_VEL
LIN {X 0,Y 93.376,Z 549.129,A -85,B 0,C 180,E1 -27278.655,E2 -27278.655} C_VEL
LIN {X 0,Y 89.828,Z 540.215,A -85,B 0,C 180,E1 -27282.054,E2 -27282.054} C_VEL
LIN {X 0,Y 88.392,Z 537.793,A -85,B 0,C 180,E1 -27283.104,E2 -27283.104} C_VEL
LIN {X 0,Y 87.013,Z 534.945,A -85,B 0,C 180,E1 -27284.249,E2 -27284.249} C_VEL
LIN {X 0,Y 86.901,Z 534.473,A -85,B 0,C 180,E1 -27284.576,E2 -27284.576} C_VEL
LIN {X 0,Y 86.587,Z 534.507,A -85,B 0,C 180,E1 -27293.941,E2 -27293.941} C_VEL
LIN {X 0,Y 86.479,Z 534.524,A -85,B 0,C 180,E1 -27299.181,E2 -27299.181} C_VEL
LIN {X 0,Y 86.533,Z 534.513,A -85,B 0,C 180,E1 -27305.691,E2 -27305.691} C_VEL
LIN {X 0,Y 86.557,Z 534.503,A -85,B 0,C 180,E1 -27313.05,E2 -27313.05} C_VEL
LIN {X 0,Y 86.551,Z 534.514,A -85,B 0,C 180,E1 -27319.488,E2 -27319.488} C_VEL
LIN {X 0,Y 86.56,Z 534.507,A -85,B 0,C 180,E1 -27325.364,E2 -27325.364} C_VEL
LIN {X 0,Y 86.583,Z 534.505,A -85,B 0,C 180,E1 -27333.231,E2 -27333.231} C_VEL
LIN {X 0,Y 86.646,Z 534.497,A -85,B 0,C 180,E1 -27341.068,E2 -27341.068} C_VEL
LIN {X 0,Y 86.967,Z 534.464,A -85,B 0,C 180,E1 -27345.969,E2 -27345.969} C_VEL
LIN {X 0,Y 87.111,Z 534.444,A -85,B 0,C 180,E1 -27350.714,E2 -27350.714} C_VEL
LIN {X 0,Y 87.723,Z 534.356,A -85,B 0,C 180,E1 -27360,E2 -27360} C_VEL
LIN {X 0,Y 87.115,Z 534.446,A -85,B 0,C 180,E1 -27369.285,E2 -27369.285} C_VEL
LIN {X 0,Y 86.947,Z 534.469,A -85,B 0,C 180,E1 -27374.087,E2 -27374.087} C_VEL
LIN {X 0,Y 86.661,Z 534.505,A -85,B 0,C 180,E1 -27378.928,E2 -27378.928} C_VEL
LIN {X 0,Y 86.582,Z 534.516,A -85,B 0,C 180,E1 -27386.767,E2 -27386.767} C_VEL
LIN {X 0,Y 86.522,Z 534.52,A -85,B 0,C 180,E1 -27395.685,E2 -27395.685} C_VEL
LIN {X 0,Y 86.516,Z 534.586,A -85,B 0,C 180,E1 -27399.852,E2 -27399.852} C_VEL
LIN {X 0,Y 86.956,Z 535.982,A -85,B 0,C 180,E1 -27401.571,E2 -27401.571} C_VEL
LIN {X 0,Y 92.017,Z 546.893,A -85,B 0,C 180,E1 -27405.609,E2 -27405.609} C_VEL
LIN {X 0,Y 94.027,Z 551.747,A -85,B 0,C 180,E1 -27407.41,E2 -27407.41} C_VEL
LIN {X 0,Y 94.495,Z 555.189,A -85,B 0,C 180,E1 -27408.394,E2 -27408.394} C_VEL
LIN {X 0,Y 94.483,Z 564.617,A -85,B 0,C 180,E1 -27411.145,E2 -27411.145} C_VEL
LIN {X 0,Y 93.923,Z 572.151,A -85,B 0,C 180,E1 -27413.692,E2 -27413.692} C_VEL
LIN {X 0,Y 92.85,Z 581.053,A -85,B 0,C 180,E1 -27417.35,E2 -27417.35} C_VEL
LIN {X 0,Y 91.719,Z 587.908,A -85,B 0,C 180,E1 -27420.762,E2 -27420.762} C_VEL
LIN {X 0,Y 89.506,Z 594.237,A -85,B 0,C 180,E1 -27424.417,E2 -27424.417} C_VEL
LIN {X 0,Y 87.479,Z 600.275,A -85,B 0,C 180,E1 -27428.809,E2 -27428.809} C_VEL
LIN {X 0,Y 85.552,Z 606.417,A -85,B 0,C 180,E1 -27434.518,E2 -27434.518} C_VEL
LIN {X 0,Y 84.414,Z 611.278,A -85,B 0,C 180,E1 -27440.417,E2 -27440.417} C_VEL
LIN {X 0,Y 84.025,Z 615.594,A -85,B 0,C 180,E1 -27447.606,E2 -27447.606} C_VEL
LIN {X 0,Y 84.082,Z 616.702,A -85,B 0,C 180,E1 -27450.002,E2 -27450.002} C_VEL
LIN {X 0,Y 84.029,Z 618.508,A -85,B 0,C 180,E1 -27454.8,E2 -27454.8} C_VEL
LIN {X 0,Y 84.395,Z 619.826,A -85,B 0,C 180,E1 -27459.59,E2 -27459.59} C_VEL
LIN {X 0,Y 85.316,Z 620.666,A -85,B 0,C 180,E1 -27464.31,E2 -27464.31} C_VEL
LIN {X 0,Y 86.772,Z 620.941,A -85,B 0,C 180,E1 -27468.906,E2 -27468.906} C_VEL
LIN {X 0,Y 88.799,Z 620.766,A -85,B 0,C 180,E1 -27473.314,E2 -27473.314} C_VEL
LIN {X 0,Y 91.34,Z 620.167,A -85,B 0,C 180,E1 -27477.497,E2 -27477.497} C_VEL
LIN {X 0,Y 94.376,Z 619.127,A -85,B 0,C 180,E1 -27481.42,E2 -27481.42} C_VEL
LIN {X 0,Y 99.907,Z 616.508,A -85,B 0,C 180,E1 -27486.725,E2 -27486.725} C_VEL
LIN {X 0,Y 104.11,Z 614.173,A -85,B 0,C 180,E1 -27489.891,E2 -27489.891} C_VEL
LIN {X 0,Y 111.168,Z 609.403,A -85,B 0,C 180,E1 -27494.063,E2 -27494.063} C_VEL
LIN {X 0,Y 116.222,Z 605.442,A -85,B 0,C 180,E1 -27496.525,E2 -27496.525} C_VEL
LIN {X 0,Y 115.069,Z 605.212,A -85,B 0,C 180,E1 -27497.791,E2 -27497.791} C_VEL
LIN {X 0,Y 110.549,Z 606.054,A -85,B 0,C 180,E1 -27500.526,E2 -27500.526} C_VEL
LIN {X 0,Y 107.047,Z 606.289,A -85,B 0,C 180,E1 -27503.781,E2 -27503.781} C_VEL
LIN {X 0,Y 103.269,Z 606.945,A -85,B 0,C 180,E1 -27507.014,E2 -27507.014} C_VEL
LIN {X 0,Y 96.181,Z 607.886,A -85,B 0,C 180,E1 -27518.571,E2 -27518.571} C_VEL
LIN {X 0,Y 94.874,Z 608.429,A -85,B 0,C 180,E1 -27531.48,E2 -27531.48} C_VEL
LIN {X 0,Y 101.056,Z 609.071,A -85,B 0,C 180,E1 -27547.996,E2 -27547.996} C_VEL
LIN {X 0,Y 104.202,Z 609.098,A -85,B 0,C 180,E1 -27551.674,E2 -27551.674} C_VEL
LIN {X 0,Y 106.862,Z 609.536,A -85,B 0,C 180,E1 -27555.252,E2 -27555.252} C_VEL
LIN {X 0,Y 100.03,Z 613.503,A -85,B 0,C 180,E1 -27560.567,E2 -27560.567} C_VEL
LIN {X 0,Y 94.161,Z 615.901,A -85,B 0,C 180,E1 -27566.605,E2 -27566.605} C_VEL
LIN {X 0,Y 89.41,Z 616.938,A -85,B 0,C 180,E1 -27573.383,E2 -27573.383} C_VEL
LIN {X 0,Y 87.676,Z 617.034,A -85,B 0,C 180,E1 -27576.714,E2 -27576.714} C_VEL
LIN {X 0,Y 85.488,Z 616.516,A -85,B 0,C 180,E1 -27582.274,E2 -27582.274} C_VEL
LIN {X 0,Y 83.923,Z 614.976,A -85,B 0,C 180,E1 -27588.911,E2 -27588.911} C_VEL
LIN {X 0,Y 83.574,Z 614.02,A -85,B 0,C 180,E1 -27591.689,E2 -27591.689} C_VEL
LIN {X 0,Y 82.727,Z 612.5,A -85,B 0,C 180,E1 -27595.583,E2 -27595.583} C_VEL
LIN {X 0,Y 81.278,Z 610.603,A -85,B 0,C 180,E1 -27599.404,E2 -27599.404} C_VEL
LIN {X 0,Y 78.649,Z 605.834,A -85,B 0,C 180,E1 -27607.07,E2 -27607.07} C_VEL
LIN {X 0,Y 78.502,Z 602.897,A -85,B 0,C 180,E1 -27610.856,E2 -27610.856} C_VEL
LIN {X 0,Y 78.754,Z 601.813,A -85,B 0,C 180,E1 -27612.066,E2 -27612.066} C_VEL
LIN {X 0,Y 80.637,Z 596.516,A -85,B 0,C 180,E1 -27617.412,E2 -27617.412} C_VEL
LIN {X 0,Y 83.16,Z 589.75,A -85,B 0,C 180,E1 -27622.717,E2 -27622.717} C_VEL
LIN {X 0,Y 85.885,Z 582.553,A -85,B 0,C 180,E1 -27627.066,E2 -27627.066} C_VEL
LIN {X 0,Y 87.434,Z 577.844,A -85,B 0,C 180,E1 -27629.422,E2 -27629.422} C_VEL
LIN {X 0,Y 87.858,Z 570.81,A -85,B 0,C 180,E1 -27632.863,E2 -27632.863} C_VEL
LIN {X 0,Y 87.98,Z 562.802,A -85,B 0,C 180,E1 -27636.239,E2 -27636.239} C_VEL
LIN {X 0,Y 87.551,Z 553.643,A -85,B 0,C 180,E1 -27639.599,E2 -27639.599} C_VEL
LIN {X 0,Y 86.742,Z 550.226,A -85,B 0,C 180,E1 -27641.016,E2 -27641.016} C_VEL
LIN {X 0,Y 83.932,Z 543.099,A -85,B 0,C 180,E1 -27644.136,E2 -27644.136} C_VEL
LIN {X 0,Y 81.591,Z 539.296,A -85,B 0,C 180,E1 -27646.169,E2 -27646.169} C_VEL
LIN {X 0,Y 79.958,Z 536.677,A -85,B 0,C 180,E1 -27647.586,E2 -27647.586} C_VEL
LIN {X 0,Y 79.626,Z 535.376,A -85,B 0,C 180,E1 -27648.16,E2 -27648.16} C_VEL
LIN {X 0,Y 79.484,Z 535.396,A -85,B 0,C 180,E1 -27657.845,E2 -27657.845} C_VEL
LIN {X 0,Y 79.449,Z 535.4,A -85,B 0,C 180,E1 -27667.237,E2 -27667.237} C_VEL
LIN {X 0,Y 79.466,Z 535.393,A -85,B 0,C 180,E1 -27675.03,E2 -27675.03} C_VEL
LIN {X 0,Y 79.451,Z 535.384,A -85,B 0,C 180,E1 -27682.756,E2 -27682.756} C_VEL
LIN {X 0,Y 79.482,Z 535.39,A -85,B 0,C 180,E1 -27692.15,E2 -27692.15} C_VEL
LIN {X 0,Y 79.512,Z 535.389,A -85,B 0,C 180,E1 -27699.295,E2 -27699.295} C_VEL
LIN {X 0,Y 79.839,Z 535.353,A -85,B 0,C 180,E1 -27705.525,E2 -27705.525} C_VEL
LIN {X 0,Y 79.995,Z 535.327,A -85,B 0,C 180,E1 -27709.88,E2 -27709.88} C_VEL
LIN {X 0,Y 80.651,Z 535.236,A -85,B 0,C 180,E1 -27720,E2 -27720} C_VEL
LIN {X 0,Y 79.998,Z 535.333,A -85,B 0,C 180,E1 -27730.119,E2 -27730.119} C_VEL
LIN {X 0,Y 79.763,Z 535.364,A -85,B 0,C 180,E1 -27735.327,E2 -27735.327} C_VEL
LIN {X 0,Y 79.521,Z 535.393,A -85,B 0,C 180,E1 -27740.702,E2 -27740.702} C_VEL
LIN {X 0,Y 79.48,Z 535.399,A -85,B 0,C 180,E1 -27747.847,E2 -27747.847} C_VEL
LIN {X 0,Y 79.477,Z 535.397,A -85,B 0,C 180,E1 -27755.895,E2 -27755.895} C_VEL
LIN {X 0,Y 79.486,Z 535.598,A -85,B 0,C 180,E1 -27757.505,E2 -27757.505} C_VEL
LIN {X 0,Y 80.508,Z 538.351,A -85,B 0,C 180,E1 -27758.661,E2 -27758.661} C_VEL
LIN {X 0,Y 82.057,Z 540.855,A -85,B 0,C 180,E1 -27759.967,E2 -27759.967} C_VEL
LIN {X 0,Y 85.336,Z 547.863,A -85,B 0,C 180,E1 -27763.014,E2 -27763.014} C_VEL
LIN {X 0,Y 88.064,Z 554.768,A -85,B 0,C 180,E1 -27765.91,E2 -27765.91} C_VEL
LIN {X 0,Y 88.073,Z 564.489,A -85,B 0,C 180,E1 -27769.029,E2 -27769.029} C_VEL
LIN {X 0,Y 87.398,Z 572.424,A -85,B 0,C 180,E1 -27771.946,E2 -27771.946} C_VEL
LIN {X 0,Y 86.341,Z 580.033,A -85,B 0,C 180,E1 -27775.267,E2 -27775.267} C_VEL
LIN {X 0,Y 85.129,Z 587.025,A -85,B 0,C 180,E1 -27778.94,E2 -27778.94} C_VEL
LIN {X 0,Y 83.156,Z 592.658,A -85,B 0,C 180,E1 -27782.303,E2 -27782.303} C_VEL
LIN {X 0,Y 80.873,Z 598.918,A -85,B 0,C 180,E1 -27786.982,E2 -27786.982} C_VEL
LIN {X 0,Y 78.708,Z 605.256,A -85,B 0,C 180,E1 -27793.133,E2 -27793.133} C_VEL
LIN {X 0,Y 77.428,Z 610.303,A -85,B 0,C 180,E1 -27799.543,E2 -27799.543} C_VEL
LIN {X 0,Y 76.955,Z 614.913,A -85,B 0,C 180,E1 -27807.385,E2 -27807.385} C_VEL
LIN {X 0,Y 77.027,Z 616.037,A -85,B 0,C 180,E1 -27810.003,E2 -27810.003} C_VEL
LIN {X 0,Y 76.992,Z 617.982,A -85,B 0,C 180,E1 -27815.24,E2 -27815.24} C_VEL
LIN {X 0,Y 77.416,Z 619.418,A -85,B 0,C 180,E1 -27820.464,E2 -27820.464} C_VEL
LIN {X 0,Y 78.454,Z 620.284,A -85,B 0,C 180,E1 -27825.592,E2 -27825.592} C_VEL
LIN {X 0,Y 80.089,Z 620.677,A -85,B 0,C 180,E1 -27830.552,E2 -27830.552} C_VEL
LIN {X 0,Y 82.332,Z 620.646,A -85,B 0,C 180,E1 -27835.268,E2 -27835.268} C_VEL
LIN {X 0,Y 85.092,Z 620.189,A -85,B 0,C 180,E1 -27839.709,E2 -27839.709} C_VEL
LIN {X 0,Y 88.391,Z 619.205,A -85,B 0,C 180,E1 -27843.822,E2 -27843.822} C_VEL
LIN {X 0,Y 92.229,Z 617.69,A -85,B 0,C 180,E1 -27847.564,E2 -27847.564} C_VEL
LIN {X 0,Y 98.793,Z 614.57,A -85,B 0,C 180,E1 -27852.52,E2 -27852.52} C_VEL
LIN {X 0,Y 106.21,Z 610.105,A -85,B 0,C 180,E1 -27856.712,E2 -27856.712} C_VEL
LIN {X 0,Y 106.653,Z 609.294,A -85,B 0,C 180,E1 -27857.864,E2 -27857.864} C_VEL
LIN {X 0,Y 102.037,Z 609.62,A -85,B 0,C 180,E1 -27861.692,E2 -27861.692} C_VEL
LIN {X 0,Y 98.052,Z 610.224,A -85,B 0,C 180,E1 -27865.012,E2 -27865.012} C_VEL
LIN {X 0,Y 90.205,Z 610.928,A -85,B 0,C 180,E1 -27877.074,E2 -27877.074} C_VEL
LIN {X 0,Y 89.091,Z 611.346,A -85,B 0,C 180,E1 -27895.476,E2 -27895.476} C_VEL
LIN {X 0,Y 94.403,Z 611.772,A -85,B 0,C 180,E1 -27908.563,E2 -27908.563} C_VEL
LIN {X 0,Y 98.996,Z 611.864,A -85,B 0,C 180,E1 -27914.371,E2 -27914.371} C_VEL
LIN {X 0,Y 95.522,Z 613.613,A -85,B 0,C 180,E1 -27917.116,E2 -27917.116} C_VEL
LIN {X 0,Y 89.039,Z 616.07,A -85,B 0,C 180,E1 -27923.245,E2 -27923.245} C_VEL
LIN {X 0,Y 83.674,Z 617.134,A -85,B 0,C 180,E1 -27930.263,E2 -27930.263} C_VEL
LIN {X 0,Y 79.627,Z 616.918,A -85,B 0,C 180,E1 -27938.158,E2 -27938.158} C_VEL
LIN {X 0,Y 77.155,Z 615.282,A -85,B 0,C 180,E1 -27946.779,E2 -27946.779} C_VEL
LIN {X 0,Y 76.378,Z 613.187,A -85,B 0,C 180,E1 -27953.24,E2 -27953.24} C_VEL
LIN {X 0,Y 76.447,Z 610.324,A -85,B 0,C 180,E1 -27959.624,E2 -27959.624} C_VEL
LIN {X 0,Y 77.593,Z 605.657,A -85,B 0,C 180,E1 -27967.183,E2 -27967.183} C_VEL
LIN {X 0,Y 78.754,Z 601.813,A -85,B 0,C 180,E1 -27972.066,E2 -27972.066} C_VEL
LIN {X 0,Y 79.205,Z 598.63,A -85,B 0,C 180,E1 -27975.565,E2 -27975.565} C_VEL
LIN {X 0,Y 78.664,Z 592.706,A -85,B 0,C 180,E1 -27981.273,E2 -27981.273} C_VEL
LIN {X 0,Y 78.572,Z 585.962,A -85,B 0,C 180,E1 -27986.676,E2 -27986.676} C_VEL
LIN {X 0,Y 79.706,Z 581.437,A -85,B 0,C 180,E1 -27989.488,E2 -27989.488} C_VEL
LIN {X 0,Y 80.82,Z 578.061,A -85,B 0,C 180,E1 -27991.243,E2 -27991.243} C_VEL
LIN {X 0,Y 81.358,Z 571.072,A -85,B 0,C 180,E1 -27994.953,E2 -27994.953} C_VEL
LIN {X 0,Y 81.623,Z 563.526,A -85,B 0,C 180,E1 -27998.419,E2 -27998.419} C_VEL
LIN {X 0,Y 81.378,Z 555.025,A -85,B 0,C 180,E1 -28001.841,E2 -28001.841} C_VEL
LIN {X 0,Y 78.865,Z 547.709,A -85,B 0,C 180,E1 -28005.504,E2 -28005.504} C_VEL
LIN {X 0,Y 74.601,Z 540.464,A -85,B 0,C 180,E1 -28010.129,E2 -28010.129} C_VEL
LIN {X 0,Y 72.863,Z 538.033,A -85,B 0,C 180,E1 -28011.886,E2 -28011.886} C_VEL
LIN {X 0,Y 72.391,Z 536.274,A -85,B 0,C 180,E1 -28012.728,E2 -28012.728} C_VEL
LIN {X 0,Y 72.376,Z 536.281,A -85,B 0,C 180,E1 -28019.079,E2 -28019.079} C_VEL
LIN {X 0,Y 72.335,Z 536.28,A -85,B 0,C 180,E1 -28025.655,E2 -28025.655} C_VEL
LIN {X 0,Y 72.311,Z 536.277,A -85,B 0,C 180,E1 -28032.866,E2 -28032.866} C_VEL
LIN {X 0,Y 72.358,Z 536.274,A -85,B 0,C 180,E1 -28040.985,E2 -28040.985} C_VEL
LIN {X 0,Y 72.337,Z 536.271,A -85,B 0,C 180,E1 -28044.342,E2 -28044.342} C_VEL
LIN {X 0,Y 72.39,Z 536.278,A -85,B 0,C 180,E1 -28050.959,E2 -28050.959} C_VEL
LIN {X 0,Y 72.393,Z 536.28,A -85,B 0,C 180,E1 -28057.149,E2 -28057.149} C_VEL
LIN {X 0,Y 72.733,Z 536.238,A -85,B 0,C 180,E1 -28065.065,E2 -28065.065} C_VEL
LIN {X 0,Y 72.88,Z 536.211,A -85,B 0,C 180,E1 -28068.88,E2 -28068.88} C_VEL
LIN {X 0,Y 73.578,Z 536.117,A -85,B 0,C 180,E1 -28080,E2 -28080} C_VEL
LIN {X 0,Y 72.882,Z 536.218,A -85,B 0,C 180,E1 -28091.119,E2 -28091.119} C_VEL
LIN {X 0,Y 72.583,Z 536.255,A -85,B 0,C 180,E1 -28096.886,E2 -28096.886} C_VEL
LIN {X 0,Y 72.397,Z 536.284,A -85,B 0,C 180,E1 -28102.849,E2 -28102.849} C_VEL
LIN {X 0,Y 72.374,Z 536.284,A -85,B 0,C 180,E1 -28109.083,E2 -28109.083} C_VEL
LIN {X 0,Y 72.381,Z 536.283,A -85,B 0,C 180,E1 -28112.894,E2 -28112.894} C_VEL
LIN {X 0,Y 73.466,Z 539.158,A -85,B 0,C 180,E1 -28114.402,E2 -28114.402} C_VEL
LIN {X 0,Y 74.973,Z 541.306,A -85,B 0,C 180,E1 -28115.885,E2 -28115.885} C_VEL
LIN {X 0,Y 77.367,Z 545.899,A -85,B 0,C 180,E1 -28118.424,E2 -28118.424} C_VEL
LIN {X 0,Y 81.112,Z 555.108,A -85,B 0,C 180,E1 -28123.026,E2 -28123.026} C_VEL
LIN {X 0,Y 81.969,Z 557.587,A -85,B 0,C 180,E1 -28124.242,E2 -28124.242} C_VEL
LIN {X 0,Y 81.637,Z 566.445,A -85,B 0,C 180,E1 -28127.387,E2 -28127.387} C_VEL
LIN {X 0,Y 80.778,Z 573.817,A -85,B 0,C 180,E1 -28130.404,E2 -28130.404} C_VEL
LIN {X 0,Y 79.268,Z 582.757,A -85,B 0,C 180,E1 -28134.813,E2 -28134.813} C_VEL
LIN {X 0,Y 78.354,Z 587.164,A -85,B 0,C 180,E1 -28137.444,E2 -28137.444} C_VEL
LIN {X 0,Y 75.574,Z 594.393,A -85,B 0,C 180,E1 -28142.294,E2 -28142.294} C_VEL
LIN {X 0,Y 72.788,Z 601.701,A -85,B 0,C 180,E1 -28148.775,E2 -28148.775} C_VEL
LIN {X 0,Y 70.968,Z 607.438,A -85,B 0,C 180,E1 -28155.669,E2 -28155.669} C_VEL
LIN {X 0,Y 70.134,Z 611.139,A -85,B 0,C 180,E1 -28161.358,E2 -28161.358} C_VEL
LIN {X 0,Y 69.946,Z 615.344,A -85,B 0,C 180,E1 -28170.003,E2 -28170.003} C_VEL
LIN {X 0,Y 69.943,Z 617.425,A -85,B 0,C 180,E1 -28175.77,E2 -28175.77} C_VEL
LIN {X 0,Y 70.468,Z 618.908,A -85,B 0,C 180,E1 -28181.509,E2 -28181.509} C_VEL
LIN {X 0,Y 71.648,Z 619.877,A -85,B 0,C 180,E1 -28187.117,E2 -28187.117} C_VEL
LIN {X 0,Y 73.49,Z 620.412,A -85,B 0,C 180,E1 -28192.493,E2 -28192.493} C_VEL
LIN {X 0,Y 75.963,Z 620.525,A -85,B 0,C 180,E1 -28197.558,E2 -28197.558} C_VEL
LIN {X 0,Y 78.991,Z 620.151,A -85,B 0,C 180,E1 -28202.268,E2 -28202.268} C_VEL
LIN {X 0,Y 82.589,Z 619.239,A -85,B 0,C 180,E1 -28206.564,E2 -28206.564} C_VEL
LIN {X 0,Y 86.727,Z 617.885,A -85,B 0,C 180,E1 -28210.416,E2 -28210.416} C_VEL
LIN {X 0,Y 93.708,Z 614.928,A -85,B 0,C 180,E1 -28215.441,E2 -28215.441} C_VEL
LIN {X 0,Y 98.011,Z 612.714,A -85,B 0,C 180,E1 -28217.857,E2 -28217.857} C_VEL
LIN {X 0,Y 97.002,Z 612.535,A -85,B 0,C 180,E1 -28219.303,E2 -28219.303} C_VEL
LIN {X 0,Y 92.774,Z 612.997,A -85,B 0,C 180,E1 -28222.697,E2 -28222.697} C_VEL
LIN {X 0,Y 84.139,Z 613.564,A -85,B 0,C 180,E1 -28235.315,E2 -28235.315} C_VEL
LIN {X 0,Y 82.274,Z 613.733,A -85,B 0,C 180,E1 -28255.1,E2 -28255.1} C_VEL
LIN {X 0,Y 87.58,Z 613.951,A -85,B 0,C 180,E1 -28269.236,E2 -28269.236} C_VEL
LIN {X 0,Y 90.746,Z 613.969,A -85,B 0,C 180,E1 -28273.435,E2 -28273.435} C_VEL
LIN {X 0,Y 87.818,Z 615.093,A -85,B 0,C 180,E1 -28276.181,E2 -28276.181} C_VEL
LIN {X 0,Y 82.814,Z 616.571,A -85,B 0,C 180,E1 -28281.004,E2 -28281.004} C_VEL
LIN {X 0,Y 78.214,Z 617.33,A -85,B 0,C 180,E1 -28286.698,E2 -28286.698} C_VEL
LIN {X 0,Y 73.509,Z 617.137,A -85,B 0,C 180,E1 -28295.005,E2 -28295.005} C_VEL
LIN {X 0,Y 70.231,Z 615.198,A -85,B 0,C 180,E1 -28305.53,E2 -28305.53} C_VEL
LIN {X 0,Y 69.23,Z 612.332,A -85,B 0,C 180,E1 -28314.306,E2 -28314.306} C_VEL
LIN {X 0,Y 69.621,Z 608.625,A -85,B 0,C 180,E1 -28322.366,E2 -28322.366} C_VEL
LIN {X 0,Y 70.971,Z 604.076,A -85,B 0,C 180,E1 -28329.718,E2 -28329.718} C_VEL
LIN {X 0,Y 73.228,Z 597.749,A -85,B 0,C 180,E1 -28337.319,E2 -28337.319} C_VEL
LIN {X 0,Y 75.845,Z 590.923,A -85,B 0,C 180,E1 -28343.346,E2 -28343.346} C_VEL
LIN {X 0,Y 78.825,Z 583.653,A -85,B 0,C 180,E1 -28348.208,E2 -28348.208} C_VEL
LIN {X 0,Y 79.706,Z 581.437,A -85,B 0,C 180,E1 -28349.488,E2 -28349.488} C_VEL
LIN {X 0,Y 80.473,Z 578.44,A -85,B 0,C 180,E1 -28351.212,E2 -28351.212} C_VEL
LIN {X 0,Y 80.422,Z 573.909,A -85,B 0,C 180,E1 -28353.922,E2 -28353.922} C_VEL
LIN {X 0,Y 79.409,Z 569.468,A -85,B 0,C 180,E1 -28356.689,E2 -28356.689} C_VEL
LIN {X 0,Y 77.267,Z 563.426,A -85,B 0,C 180,E1 -28360.51,E2 -28360.51} C_VEL
LIN {X 0,Y 75.17,Z 557.115,A -85,B 0,C 180,E1 -28364.205,E2 -28364.205} C_VEL
LIN {X 0,Y 73.56,Z 551.947,A -85,B 0,C 180,E1 -28367.172,E2 -28367.172} C_VEL
LIN {X 0,Y 69.763,Z 545.244,A -85,B 0,C 180,E1 -28372.116,E2 -28372.116} C_VEL
LIN {X 0,Y 68.106,Z 542.187,A -85,B 0,C 180,E1 -28374.494,E2 -28374.494} C_VEL
LIN {X 0,Y 65.894,Z 539.293,A -85,B 0,C 180,E1 -28377.275,E2 -28377.275} C_VEL
LIN {X 0,Y 65.317,Z 537.161,A -85,B 0,C 180,E1 -28378.519,E2 -28378.519} C_VEL
LIN {X 0,Y 65.214,Z 537.171,A -85,B 0,C 180,E1 -28382.601,E2 -28382.601} C_VEL
LIN {X 0,Y 65.247,Z 537.161,A -85,B 0,C 180,E1 -28391.061,E2 -28391.061} C_VEL
LIN {X 0,Y 65.265,Z 537.163,A -85,B 0,C 180,E1 -28399.751,E2 -28399.751} C_VEL
LIN {X 0,Y 65.258,Z 537.169,A -85,B 0,C 180,E1 -28409.487,E2 -28409.487} C_VEL
LIN {X 0,Y 65.244,Z 537.165,A -85,B 0,C 180,E1 -28414.476,E2 -28414.476} C_VEL
LIN {X 0,Y 65.634,Z 537.122,A -85,B 0,C 180,E1 -28424.506,E2 -28424.506} C_VEL
LIN {X 0,Y 65.772,Z 537.098,A -85,B 0,C 180,E1 -28427.66,E2 -28427.66} C_VEL
LIN {X 0,Y 66.502,Z 536.997,A -85,B 0,C 180,E1 -28440,E2 -28440} C_VEL
LIN {X 0,Y 65.781,Z 537.102,A -85,B 0,C 180,E1 -28452.338,E2 -28452.338} C_VEL
LIN {X 0,Y 65.387,Z 537.156,A -85,B 0,C 180,E1 -28458.81,E2 -28458.81} C_VEL
LIN {X 0,Y 65.285,Z 537.302,A -85,B 0,C 180,E1 -28467.173,E2 -28467.173} C_VEL
LIN {X 0,Y 66.335,Z 540.014,A -85,B 0,C 180,E1 -28468.926,E2 -28468.926} C_VEL
LIN {X 0,Y 68.23,Z 542.441,A -85,B 0,C 180,E1 -28471.214,E2 -28471.214} C_VEL
LIN {X 0,Y 71.867,Z 549.098,A -85,B 0,C 180,E1 -28475.926,E2 -28475.926} C_VEL
LIN {X 0,Y 74.332,Z 555.54,A -85,B 0,C 180,E1 -28479.658,E2 -28479.658} C_VEL
LIN {X 0,Y 75.798,Z 559.974,A -85,B 0,C 180,E1 -28482.122,E2 -28482.122} C_VEL
LIN {X 0,Y 74.933,Z 570.818,A -85,B 0,C 180,E1 -28486.615,E2 -28486.615} C_VEL
LIN {X 0,Y 73.347,Z 579.503,A -85,B 0,C 180,E1 -28490.931,E2 -28490.931} C_VEL
LIN {X 0,Y 71.653,Z 587.2,A -85,B 0,C 180,E1 -28495.672,E2 -28495.672} C_VEL
LIN {X 0,Y 68.661,Z 594.368,A -85,B 0,C 180,E1 -28500.912,E2 -28500.912} C_VEL
LIN {X 0,Y 65.71,Z 601.634,A -85,B 0,C 180,E1 -28508.02,E2 -28508.02} C_VEL
LIN {X 0,Y 64.136,Z 606.296,A -85,B 0,C 180,E1 -28514.104,E2 -28514.104} C_VEL
LIN {X 0,Y 62.928,Z 611.781,A -85,B 0,C 180,E1 -28523.591,E2 -28523.591} C_VEL
LIN {X 0,Y 62.887,Z 614.637,A -85,B 0,C 180,E1 -28530.003,E2 -28530.003} C_VEL
LIN {X 0,Y 62.917,Z 616.785,A -85,B 0,C 180,E1 -28536.417,E2 -28536.417} C_VEL
LIN {X 0,Y 63.557,Z 618.356,A -85,B 0,C 180,E1 -28542.78,E2 -28542.78} C_VEL
LIN {X 0,Y 64.91,Z 619.464,A -85,B 0,C 180,E1 -28548.958,E2 -28548.958} C_VEL
LIN {X 0,Y 66.982,Z 620.145,A -85,B 0,C 180,E1 -28554.819,E2 -28554.819} C_VEL
LIN {X 0,Y 69.742,Z 620.369,A -85,B 0,C 180,E1 -28560.259,E2 -28560.259} C_VEL
LIN {X 0,Y 73.074,Z 620.039,A -85,B 0,C 180,E1 -28565.247,E2 -28565.247} C_VEL
LIN {X 0,Y 77.007,Z 619.278,A -85,B 0,C 180,E1 -28569.71,E2 -28569.71} C_VEL
LIN {X 0,Y 81.471,Z 618.08,A -85,B 0,C 180,E1 -28573.642,E2 -28573.642} C_VEL
LIN {X 0,Y 87.727,Z 615.804,A -85,B 0,C 180,E1 -28577.983,E2 -28577.983} C_VEL
LIN {X 0,Y 88.318,Z 615.267,A -85,B 0,C 180,E1 -28579.403,E2 -28579.403} C_VEL
LIN {X 0,Y 78.014,Z 615.736,A -85,B 0,C 180,E1 -28593.229,E2 -28593.229} C_VEL
LIN {X 0,Y 75.319,Z 615.694,A -85,B 0,C 180,E1 -28614.646,E2 -28614.646} C_VEL
LIN {X 0,Y 82.112,Z 615.653,A -85,B 0,C 180,E1 -28632.284,E2 -28632.284} C_VEL
LIN {X 0,Y 79.872,Z 616.438,A -85,B 0,C 180,E1 -28635.306,E2 -28635.306} C_VEL
LIN {X 0,Y 73.092,Z 617.532,A -85,B 0,C 180,E1 -28642.62,E2 -28642.62} C_VEL
LIN {X 0,Y 70.53,Z 617.683,A -85,B 0,C 180,E1 -28646.252,E2 -28646.252} C_VEL
LIN {X 0,Y 66.936,Z 617.238,A -85,B 0,C 180,E1 -28652.858,E2 -28652.858} C_VEL
LIN {X 0,Y 63.973,Z 615.825,A -85,B 0,C 180,E1 -28661.236,E2 -28661.236} C_VEL
